# B&R Automation Studio project dbserv_0640
Automation Studio 6.5.3.11

## Configuration CP3686X

CPU X20CP3686X, AutomationRuntime 6.7.6, Build 11.3.0

### Task classes (Cpu.sw)
```
Cyclic#3:
  io <- IO-Treiber.io.prg
  kupplung <- Anwendung.kupplung.prg
  anlage <- Anwendung.anlage.prg
  iec103 <- IEC103-Treiber.iec103.prg
  iodrv <- IO-Treiber.iodrv.prg
  dbsevent <- DbServ-Basis.dbsevent.prg
  iec103Cmd <- IEC103-Treiber.iec103Cmd.prg
Cyclic#4:
  def <- def.prg
  Lebensbit <- Lebensbit.prg
  zaehler <- zaehler.prg
Cyclic#8:
  dbstcp <- DbServ-Basis.dbstcp.prg
  dbserv <- DbServ-Basis.dbserv.prg
  dbsmon <- DbServ-Basis.dbsmon.prg
  dbstest <- DbServ-Basis.dbstest.prg
DataObjects: dplist <- Anwendung.dplist.dob, typlist <- Anwendung.typlist.dob
Binaries: TCData, udbdef, sysconf, iomap, asfw, arconfig, ashwd, ashwac, mvLoader
Libraries: dbslib, sys_lib, standard, runtime, OPERATOR, FileIO, dvframe, DPMaster, DataObj, CAN_Lib, brsystem, astime, AsHW, AsBrStr, IEC103Ut, ArEventLog, AsIecCon, ethsock
```

### Hardware
```
PLC1 : X20CP3686X v1.10.0.0
  Connector IF2:
    ActivateDevice = 1
    HostName = audiinba6183
    Mode = Manual
    InternetAddress = 192.168.0.86
    SubnetMask = 255.255.255.0
    ActivateSnmp = 2
  Connector IF3:
    CycleTime = 2000
    InaPort = 11161
    InaNodeNumber = 0
  ConfigurationID = dbserv86_Config1
  UserPartitionSize = 0
  UserRamSize = 966656
  RemMemSize = 65280
  VolatileGlobalPvSize = 4096
  XLinkUseDefault = 0
  XLinkDuration = 10000
  FileDevice1
  FileDeviceName1 = USER
  FileDevicePath1 = USER_PATH
  EthernetHostName = DbServ
  EthernetDefaultGateway = 255.255.255.255
  ActivateWebServer = 0
  ActivateSdm = 0
  ActivateFtpServer = 1
X20BM11 : X20BM11 v1.1.0.0 (Disabled=true)  [X2X1 -> PLC1.IF6]
X20CS1030 : X20CS1030 v1.8.3.0 (Disabled=true)  [SS1 -> X20TB12.SS; SL -> X20BM11.SL1]
X20TB12 : X20TB12 v1.0.0.0 (Disabled=true)
```

### ACTIVE_GDM.osl - PLC1/States/ACTIVE_GDM.osl
```
ObjectStates:
  Object io (Memory=UserROM, Enable=true)
  Object zaehler (Memory=UserROM, Enable=false)
  Object kupplung (Memory=UserROM, Enable=true)
  Object iec103 (Memory=UserROM, Enable=true)
  Object iodrv (Memory=UserROM, Enable=true)
  Object l2dp (Memory=UserROM, Enable=true)
  Object dbsevent (Memory=UserROM, Enable=false)
  Object battery (Memory=UserROM, Enable=true)
  Object dbserv (Memory=UserROM, Enable=true)
  Object dbsmon (Memory=UserROM, Enable=true)
  Object dbstest (Memory=UserROM, Enable=false)
  Object dbstcp (Memory=UserROM, Enable=true)
  Object dbvist (Memory=UserROM, Enable=true)
  Object dbvisint (Memory=UserROM, Enable=true)
  Object gps (Memory=UserROM, Enable=true)
  Object version (Memory=UserROM, Enable=true)
  Object ydplist (Memory=UserROM, Enable=false)
  Object ytyplist (Memory=UserROM, Enable=false)
  Object dplist1 (Memory=UserROM, Enable=false)
  Object typlist1 (Memory=UserROM, Enable=false)
  Object dplist (Memory=UserROM, Enable=true)
  Object typlist (Memory=UserROM, Enable=true)
  Object dplisto (Memory=UserROM, Enable=false)
  Object ioimgcfg (Memory=UserROM, Enable=true)
  Object a_rflx_io (Memory=UserROM, Enable=true)
  Object dbv_text (Memory=UserROM, Enable=true)
  Object dbv_par (Memory=UserROM, Enable=true)
  Object dbv_env (Memory=UserROM, Enable=true)
  Object dbv_atoa (Memory=UserROM, Enable=true)
  Object dbv_func (Memory=UserROM, Enable=true)
  Object dbv_code (Memory=UserROM, Enable=true)
  Object dbv_rs (Memory=UserROM, Enable=true)
  Object dbv_vt1 (Memory=UserROM, Enable=true)
  Object dpm_099 (Memory=UserROM, Enable=true)
  Object sysconf (Memory=SystemROM, Enable=true)
  Object String_x (Memory=UserROM, Enable=true)
  Object megafubs (Memory=UserROM, Enable=true)
  Object dbv_lib (Memory=UserROM, Enable=true)
  Object dbvi_lib (Memory=UserROM, Enable=true)
  Object dbslib (Memory=UserROM, Enable=true)
  Object DA_x (Memory=UserROM, Enable=true)
```

## Logical view

Binary libraries used (declarations not repeated): ETHSOCK, sys_lib, runtime, standard, operator, FileIO, dvframe, DPMaster, DataObj, CAN_Lib, brsystem, astime, AsBrStr, AsHW, ArEventLog, AsIecCon

### Data object Logical/version (Simple, version 6.00.0) - Softwarestand

#### version.dat
```
; durchgeführte Software-Änderungen

;	14.07.2023	BIE     Version 6.40.0 		Kompiliert mit AS 4.12.3
;											für ATOM-CPUs mit AR E4.93

;	08.11.2021	BIE     Version 6.30.0 		Bugfix in Modul dbserv.c

;	15.07.2021	BIE     Version 6.20.0 		Kompiliert mit AS 4.9.3
;											für ATOM-CPUs mit AR D4.90
;											CELERON-CPUs werden nicht mehr unterstützt

;	02.03.2020	BIE     Version 6.11.0 		Kompiliert mit AS 4.6.4
;											für ATOM-CPUs mit AR C4.63
;											für CELERON-CPUs mit AR H3.10

;	04.12.2019	BIE     Version 6.10.0 		Kompiliert mit AS 4.4.6
;											für ATOM-CPUs mit AR C4.45
;											Lib IEC103Ut für IEC-Kommandos wurde hinzugefügt
;											dbseventtreiber aktualisiert
;
;	08.03.2019	BIE     Version 6.00.0 		Kompiliert mit AS 4.4.6
;											für ATOM-CPUs mit AR G4.34
;
;   12.10.2016	BIE     Version 4.11.0 		Kompiliert mit AS 4.1.11
;											Der angepasste IEC-Treiber von WAI wurde hinzugefügt und der dbsevent Treiber von KRZ
;											Ausserdem werden nun zwei Versionen der .br-Module veröffentlicht:
;											4.11.0 für ATOM-CPUs mit AR E4.10
;											3.11.0 für ATOM-CPUs mit AR V3.09

;   31.07.15	BIE     Version 4.10.0 		Portierung in AS 4.1.6.81 mit AR E4.10
;											inkl. Anpassungen für dbtcp für ATOM CPUs mit AR >x4.xx
;
;	12.08.13	WAI		Version 3.00.0		diverse Tests, Bereinigung der Sourcecodes
;
;	29.07.13	KRZ		Version 3.00.0		Portierung auf AS 3.0.90.23 SP05
;
;	30.06.11	RES		Version 2.07.1		Entwicklungsprojekt und Beispielprojekt mit AS2.7 kompiliert
;											AS V 2.7.0.20 SP13
;											AR N 2.95
;											Keine funktionellen Aenderungen
;
;	18.01.11	RES		Version 2.07		Erste freigegebene Vollversion für X20 CPUs
;						dbserv86.pgp		Neues Entwicklungsprojekt mit X20CP3486 erstellt
;											AS V 2.6.0.7
;											AR V 2.92
;						dbsbs486.pgp		Neues Beispielprojekt für X20CP3486 erstellt
;											AS + AR wie oben
;											Keine funktionellen Aenderungen
;
;	26.11.10	WAI		Version 2.06.4
;						iec103		IsANumber() geaendert: nun mit Vorzeichen Unterstuetzung
;						iodrv		Schreibzugriff auf PVs aktiviert
;
;	04.11.09	WAI		Version 2.06.3
;						l2dp		um510.c	verbesserte Reihenfolge beim Polling der Profile wegen Probleme bei langsamen Reaktionszeiten
;
;	12.10.09	WAI		Version 2.06.2
;						l2dp		neues Schlüsselwort Endian (=Big oder =Little) für Byte-Order
;									Profibus-Diagnose pL2DP_PbDataIn jetzt 244 statt 128 Byte
;
;	01.10.09	WAI		Version 2.06.1
;						l2dp		neues Schlüsselwort Inv (Invers) für BOOL-Variablen
;
;	21.08.09	WAI		Version 2.06 alle Module gestempelt
;						l2dp		neue Device-Variante UMG510
;									neue Schlüsselworte für GSD-Treiber (Mode, ModePar) wegen SYMAP
;
;	21.04.08	WAI		Version 2.05
;						l2dp		neue Device-Variante SPAZC302 für ABB-Gateways
;
;	20.02.08	WAI		Version 2.04
;						l2dp		neue Device-Variante UMGProfil für UMG96S und UMG507
;
;	28.01.08	RES		Version 2.04
;						dbslib:		Fehlerbehebung durch KUR: Status bei DbsGetBool() und DbsGetInt()
;						dbvi_lib:	Fehlerbehebung durch KUR: Output-Aktualisierung in letzter Displayzeile
;
;	25.06.07	WAI		Version 2.03 für IEC-Treiber (Anpassung Mode 13)
;
;	18.05.07	WAI		Version 2.02
;						dbsmon.c	Anzeige des valid-Status
;						gsd.c,l2dp.h,l2dp_parse.c,l2dp_parse.h
;									neuer Profibus-Typ "GSD"
;									jetzt 4 statt 1 L2DP-Linie möglich, dafür aber max. 64 statt 128 devices per line
;									(wegen 64kB-Grenze)
;						dbv_text.dat negative Werte ermöglicht incl. Korrektur bei Nachkommastellen
;						dbvist.c	Alarmquittierung aktiviert (direktes Schreiben in PAB)
;						alle anderen Module:	ebenfalls auf V2.02 gestempelt, um Verwirrungen zu vermeiden
;
;	09.05.07	WAI		Version 2.01 (Projektabgleich)
;						l2dp.c		Defaultwert Fakt = 1.0
;						umg503.c	kein neuer Request bei Kopplungsstörung wegen wiederholten Fehlermeldungen
;						iodrv.c		Schreibattribut für quittierpflichtige Variablen
;						dbv_rs.dat	9600Bd wegen Problem mit IF060 und Tableau
;
;	08.09.06	WAI		Version 2.00
;	04.07.06	WAI		Version mit neuem DbVist
;	22.06.06	WAI		Version mit DbVist
;	07.04.06	WAI		Erstfassung
```

### Global.typ
```iecst
TYPE
	XstDiagnose : 	STRUCT
		ulFRM_rbufFailAnz : UDINT;
		ulFRM_readFailAnz : UDINT;
		ulWrongTelAnz : UDINT;
		ulDTExSetTimeFail : UDINT;
		ulTelTimeoutAnz : UDINT;
		ulSyncAnz : UDINT;
		ulRTC_gettimeFail : UDINT;
		ulSyncPosFail : UDINT;
	END_STRUCT;
	XstMeinberg : 	STRUCT
		ucTag : USINT;
		ucMonat : USINT;
		ucJahr : USINT;
		ucStunden : USINT;
		ucMinuten : USINT;
		ucSekunden : USINT;
		ucSyncOK : USINT;
		ucPosOK : USINT;
		ucZZone : USINT;
		ucZSprung : USINT;
	END_STRUCT;
END_TYPE
```

### Library Logical/Libraries/IEC103Ut (IEC, version 6.40.0)

#### IEC103Ut.typ - Exported data types
```iecst
TYPE
	IEC103Ut_WrCmd_PVInfo_Type : 	STRUCT
		PVAdr : UDINT;
		PVLen : UDINT;
		PVDataType : UDINT;
		PVDimension : UINT;
	END_STRUCT;
END_TYPE
```

#### IEC103Ut.var - Exported constants
```iecst
VAR CONSTANT
	IEC103Ut_DATA_TYPE_STRUCT : USINT := 0;
	IEC103Ut_DATA_TYPE_STRUCT_2 : USINT := 15;
	IEC103Ut_DATA_TYPE_BOOL : USINT := 1;
	IEC103Ut_DATA_TYPE_SINT : USINT := 2;
	IEC103Ut_DATA_TYPE_INT : USINT := 3;
	IEC103Ut_DATA_TYPE_DINT : USINT := 4;
	IEC103Ut_DATA_TYPE_USINT : USINT := 5;
	IEC103Ut_DATA_TYPE_UINT : USINT := 6;
	IEC103Ut_DATA_TYPE_UDINT : USINT := 7;
	IEC103Ut_DATA_TYPE_REAL : USINT := 8;
	IEC103Ut_DATA_TYPE_STRING : USINT := 9;
	IEC103Ut_DATA_TYPE_ULINT : USINT := 10;
	IEC103Ut_DATA_TYPE_DATE_AND_TIME : USINT := 11;
	IEC103Ut_DATA_TYPE_TIME : USINT := 12;
	IEC103Ut_DATA_TYPE_DATE : USINT := 13;
	IEC103Ut_DATA_TYPE_LREAL : USINT := 14;
END_VAR
(**)
VAR CONSTANT
	IEC103Ut_FUB_IDLE : DINT := 65533;
	IEC103Ut_FUB_DISABLED : DINT := 65534;
	IEC103Ut_FUB_BUSY : DINT := 65535;
	IED103Ut_ERROR_START : DINT := 50000;
	IED103Ut_ERROR_INPUT_INVALID : DINT := IED103Ut_ERROR_START+2000;
END_VAR
```

#### IEC103Ut.fun - Exported functions and function blocks
```iecst
{REDUND_ERROR} FUNCTION_BLOCK IEC103Ut_WrCmd (*TODO: Hier einen Kommentar eingeben*) (*$GROUP=User,$CAT=User,$GROUPICON=User.png,$CATICON=User.png*)
	VAR_INPUT
		Enable : BOOL;
		DataSend : BOOL;
		LineVarStr : UDINT;
		LineNumber : USINT;
		DeviceAdr : USINT;
		FunctionType : USINT;
		InformationNumber : USINT;
		Val : USINT;
	END_VAR
	VAR_OUTPUT
		Status : DINT;
	END_VAR
	VAR
		WrCmdStep : UINT;
		PVStr : STRING[100];
		ValStr : STRING[10];
		ItemStr : STRING[100];
		PV_xgetadr_status : UINT;
		PV_ninfo_status : UINT;
		PVInfo_AnlStruct : IEC103Ut_WrCmd_PVInfo_Type;
		PVInfo_AnlStructOld : IEC103Ut_WrCmd_PVInfo_Type;
		PVInfo_DataSend : IEC103Ut_WrCmd_PVInfo_Type;
		PVInfo_DeviceAdress : IEC103Ut_WrCmd_PVInfo_Type;
		PVInfo_FunctionType : IEC103Ut_WrCmd_PVInfo_Type;
		PVInfo_InformationNumber : IEC103Ut_WrCmd_PVInfo_Type;
		PVInfo_Val : IEC103Ut_WrCmd_PVInfo_Type;
		PVInfo_Ready : IEC103Ut_WrCmd_PVInfo_Type;
		PVInfo_Error : IEC103Ut_WrCmd_PVInfo_Type;
		IECIEC103Ut_WrSimplePV_0 : IEC103Ut_WrSimplePV;
		IEC103Ut_RdSimplePV_0 : IEC103Ut_RdSimplePV;
		LineVarStrOld : UDINT;
		LineNumberOld : USINT;
	END_VAR
END_FUNCTION_BLOCK

{REDUND_ERROR} FUNCTION_BLOCK IEC103Ut_WrSimplePV (*TODO: Hier einen Kommentar eingeben*) (*$GROUP=User,$CAT=User,$GROUPICON=User.png,$CATICON=User.png*)
	VAR_INPUT
		PVAdr : {REDUND_UNREPLICABLE} UDINT;
		DataType : UDINT;
		PVValue : DINT;
	END_VAR
	VAR_OUTPUT
		valid : BOOL;
	END_VAR
	VAR
		pPV_BOOL : REFERENCE TO BOOL;
		pPV_USINT : REFERENCE TO USINT;
		pPV_UINT : REFERENCE TO UINT;
		pPV_UDINT : REFERENCE TO UDINT;
		pPV_SINT : REFERENCE TO SINT;
		pPV_INT : REFERENCE TO INT;
		pPV_DINT : REFERENCE TO DINT;
		pPV_REAL : REFERENCE TO REAL;
	END_VAR
END_FUNCTION_BLOCK

{REDUND_ERROR} FUNCTION_BLOCK IEC103Ut_RdSimplePV (*TODO: Hier einen Kommentar eingeben*) (*$GROUP=User,$CAT=User,$GROUPICON=User.png,$CATICON=User.png*)
	VAR_INPUT
		PVAdr : {REDUND_UNREPLICABLE} UDINT;
		DataType : UDINT;
	END_VAR
	VAR_OUTPUT
		PVValue : DINT;
		valid : BOOL;
	END_VAR
	VAR
		pPV_BOOL : REFERENCE TO BOOL;
		pPV_USINT : REFERENCE TO USINT;
		pPV_UINT : REFERENCE TO UINT;
		pPV_UDINT : REFERENCE TO UDINT;
		pPV_SINT : REFERENCE TO SINT;
		pPV_INT : REFERENCE TO INT;
		pPV_DINT : REFERENCE TO DINT;
		pPV_REAL : REFERENCE TO REAL;
	END_VAR
END_FUNCTION_BLOCK
```

#### IEC103Ut_WrCmd.st
```iecst
(*
-----------------------------------------------
FUNCTION Block IEC103Ut_WrCmd

	Write commands to a device, using the command structure OF IEC103 Task

	Inputs:
		Enable		 		Enable function block
		DataSend			Send command do device (edge sensitive)
		LineVarStr			Option: Adress OF name OF local PV structure element in Task IEC103 (example: "iec103:stANL[0].Command")
		LineNumber			Option:	Linenumber (1..12)
							Either LineVarStr or LineNumber is necessary
		DeviceAdr			Adress of device
		FunctionType		Function Type
		InformationNumber	Information Number
		Val					Value

	Outputs:
		Status				0 		Function ready, without error

							52000	Invalid input parameter
							52008	Timeout response telegram
							52020	command NOT accepted
							52023	response telegram: value not equal
							52024	response telegram: return information not equal
							52025	command function disabled
							52026	connection to device not ready
							52027	wrong device adress
							52028	command function still active

							3300 - 14714	error state of function PV_xgetadr or PV_ninfo (see B&R Help)

							65533	functionblock idle
							65534	functionblock disabled
							65535	functionblock busy

	Version:
	07.02.2019	Version 1.0
				first edition

-----------------------------------------------
*)
FUNCTION_BLOCK IEC103Ut_WrCmd

	IF(Enable = TRUE) THEN
		CASE WrCmdStep OF
			0:
				// ---------------------
				// check input parameter
				IF((LineVarStr = 0) AND (LineNumber = 0)) THEN
					Status		:= IED103Ut_ERROR_INPUT_INVALID;
					WrCmdStep	:= 210;
				ELSE

					Status := IEC103Ut_FUB_BUSY;
					// ---------------------------------------------
					// get name and adress of main structure element
					IF(LineVarStr = 0) THEN
						// Adresse der Anlagenstruktur ermitteln: PV Name erzeugen und PV Adresse ermitteln
						brsstrcpy(ADR(PVStr),ADR('iec103:stANL['));
						brsitoa(USINT_TO_DINT(LineNumber-1),ADR(ValStr));
						brsstrcat(ADR(PVStr),ADR(ValStr));
						brsstrcat(ADR(PVStr),ADR('].Command'));
					ELSE
						// Adresse der Anlagenstruktur ermitteln: Uebergebenen PV Namen verwenden und PV Adresse ermitteln
						brsstrcpy(ADR(PVStr),LineVarStr);
					END_IF

					PV_xgetadr_status := PV_xgetadr(ADR(PVStr),ADR(PVInfo_AnlStruct.PVAdr),ADR(PVInfo_AnlStruct.PVLen));

					IF(PV_xgetadr_status = 0) THEN
						LineNumberOld	:= LineNumber;
						LineVarStrOld	:= LineVarStr;
						WrCmdStep		:= 10;
					ELSE
						Status			:= PV_xgetadr_status;
						WrCmdStep		:= 210;
					END_IF
				END_IF

			10:	// get adress and info about structure element: DataSend
				brsstrcpy(ADR(ItemStr),ADR(PVStr));
				brsstrcat(ADR(ItemStr),ADR('.DataSend'));
				PV_xgetadr_status := PV_xgetadr(ADR(ItemStr),ADR(PVInfo_DataSend.PVAdr),ADR(PVInfo_DataSend.PVLen));
				IF(PV_xgetadr_status = 0) THEN
					WrCmdStep	:= 11;
				ELSE
					Status		:= PV_xgetadr_status;
					WrCmdStep	:= 210;
				END_IF

			11:
				PV_ninfo_status := PV_ninfo(ADR(ItemStr),ADR(PVInfo_DataSend.PVDataType),ADR(PVInfo_DataSend.PVLen),ADR(PVInfo_DataSend.PVDimension));
				IF(PV_ninfo_status = 0) THEN
					WrCmdStep	:= 15;
				ELSE
					Status		:= PV_ninfo_status;
					WrCmdStep	:= 210;
				END_IF

			15:	// get adress and info about structure element: PVInfo_DeviceAdress
				brsstrcpy(ADR(ItemStr),ADR(PVStr));
				brsstrcat(ADR(ItemStr),ADR('.DeviceAdress'));
				PV_xgetadr_status := PV_xgetadr(ADR(ItemStr),ADR(PVInfo_DeviceAdress.PVAdr),ADR(PVInfo_DeviceAdress.PVLen));
				IF(PV_xgetadr_status = 0) THEN
					WrCmdStep	:= 16;
				ELSE
					Status		:= PV_xgetadr_status;
					WrCmdStep	:= 210;
				END_IF

			16:
				PV_ninfo_status := PV_ninfo(ADR(ItemStr),ADR(PVInfo_DeviceAdress.PVDataType),ADR(PVInfo_DeviceAdress.PVLen),ADR(PVInfo_DeviceAdress.PVDimension));
				IF(PV_ninfo_status = 0) THEN
					WrCmdStep	:= 20;
				ELSE
					Status		:= PV_ninfo_status;
					WrCmdStep	:= 210;
				END_IF

			20:	// get adress and info about structure element: FunctionType
				brsstrcpy(ADR(ItemStr),ADR(PVStr));
				brsstrcat(ADR(ItemStr),ADR('.FunctionType'));
				PV_xgetadr_status := PV_xgetadr(ADR(ItemStr),ADR(PVInfo_FunctionType.PVAdr),ADR(PVInfo_FunctionType.PVLen));
				IF(PV_xgetadr_status = 0) THEN
					WrCmdStep	:= 21;
				ELSE
					Status		:= PV_xgetadr_status;
					WrCmdStep	:= 210;
				END_IF

			21:
				PV_ninfo_status := PV_ninfo(ADR(ItemStr),ADR(PVInfo_FunctionType.PVDataType),ADR(PVInfo_FunctionType.PVLen),ADR(PVInfo_FunctionType.PVDimension));
				IF(PV_ninfo_status = 0) THEN
					WrCmdStep	:= 25;
				ELSE
					Status		:= PV_ninfo_status;
					WrCmdStep	:= 210;
				END_IF

			25:	// get adress and info about structure element: InformationNumber
				brsstrcpy(ADR(ItemStr),ADR(PVStr));
				brsstrcat(ADR(ItemStr),ADR('.InformationNumber'));
				PV_xgetadr_status := PV_xgetadr(ADR(ItemStr),ADR(PVInfo_InformationNumber.PVAdr),ADR(PVInfo_InformationNumber.PVLen));
				IF(PV_xgetadr_status = 0) THEN
					WrCmdStep	:= 26;
				ELSE
					Status		:= PV_xgetadr_status;
					WrCmdStep	:= 210;
				END_IF

			26:
				PV_ninfo_status := PV_ninfo(ADR(ItemStr),ADR(PVInfo_InformationNumber.PVDataType),ADR(PVInfo_InformationNumber.PVLen),ADR(PVInfo_InformationNumber.PVDimension));
				IF(PV_ninfo_status = 0) THEN
					WrCmdStep	:= 30;
				ELSE
					Status		:= PV_ninfo_status;
					WrCmdStep	:= 210;
				END_IF

			30:	// get adress and info about structure element: Val
				brsstrcpy(ADR(ItemStr),ADR(PVStr));
				brsstrcat(ADR(ItemStr),ADR('.Val'));
				PV_xgetadr_status := PV_xgetadr(ADR(ItemStr),ADR(PVInfo_Val.PVAdr),ADR(PVInfo_Val.PVLen));
				IF(PV_xgetadr_status = 0) THEN
					WrCmdStep	:= 31;
				ELSE
					Status		:= PV_xgetadr_status;
					WrCmdStep	:= 210;
				END_IF

			31:
				PV_ninfo_status := PV_ninfo(ADR(ItemStr),ADR(PVInfo_Val.PVDataType),ADR(PVInfo_Val.PVLen),ADR(PVInfo_Val.PVDimension));
				IF(PV_ninfo_status = 0) THEN
					WrCmdStep	:= 35;
				ELSE
					Status		:= PV_ninfo_status;
					WrCmdStep	:= 210;
				END_IF

			35:	// get adress and info about structure element: Ready
				brsstrcpy(ADR(ItemStr),ADR(PVStr));
				brsstrcat(ADR(ItemStr),ADR('.Ready'));
				PV_xgetadr_status := PV_xgetadr(ADR(ItemStr),ADR(PVInfo_Ready.PVAdr),ADR(PVInfo_Ready.PVLen));
				IF(PV_xgetadr_status = 0) THEN
					WrCmdStep	:= 36;
				ELSE
					Status		:= PV_xgetadr_status;
					WrCmdStep	:= 210;
				END_IF

			36:
				PV_ninfo_status := PV_ninfo(ADR(ItemStr),ADR(PVInfo_Ready.PVDataType),ADR(PVInfo_Ready.PVLen),ADR(PVInfo_Ready.PVDimension));
				IF(PV_ninfo_status = 0) THEN
					WrCmdStep	:= 40;
				ELSE
					Status		:= PV_ninfo_status;
					WrCmdStep	:= 210;
				END_IF

			40:	// get adress and info about structure element: Error
				brsstrcpy(ADR(ItemStr),ADR(PVStr));
				brsstrcat(ADR(ItemStr),ADR('.Error'));
				PV_xgetadr_status := PV_xgetadr(ADR(ItemStr),ADR(PVInfo_Error.PVAdr),ADR(PVInfo_Error.PVLen));
				IF(PV_xgetadr_status = 0) THEN
					WrCmdStep	:= 41;
				ELSE
					Status		:= PV_xgetadr_status;
					WrCmdStep	:= 210;
				END_IF

			41:
				PV_ninfo_status := PV_ninfo(ADR(ItemStr),ADR(PVInfo_Error.PVDataType),ADR(PVInfo_Error.PVLen),ADR(PVInfo_Error.PVDimension));
				IF(PV_ninfo_status = 0) THEN
					WrCmdStep	:= 100;
				ELSE
					Status		:= PV_ninfo_status;
					WrCmdStep	:= 210;
				END_IF

			100:
				// Idle step, wait for command to send
				IF(DataSend = TRUE) THEN
					IF((LineNumberOld <> LineNumber) OR (LineVarStrOld <> LineVarStr)) THEN
						Status		:= IEC103Ut_FUB_BUSY;
						WrCmdStep	:= 0;
					ELSE
						IF(DeviceAdr = 0) THEN
							Status		:= IED103Ut_ERROR_INPUT_INVALID;
							WrCmdStep	:= 120;
						ELSE
							// Send command to device
							Status := IEC103Ut_FUB_BUSY;

							// Write parameter and command to local structure of iec task
							IECIEC103Ut_WrSimplePV_0(PVAdr := PVInfo_Ready.PVAdr, 				DataType := PVInfo_Ready.PVDataType,				PVValue := 0);
							IECIEC103Ut_WrSimplePV_0(PVAdr := PVInfo_FunctionType.PVAdr,		DataType := PVInfo_FunctionType.PVDataType,			PVValue := FunctionType);
							IECIEC103Ut_WrSimplePV_0(PVAdr := PVInfo_InformationNumber.PVAdr,	DataType := PVInfo_InformationNumber.PVDataType,	PVValue := InformationNumber);
							IECIEC103Ut_WrSimplePV_0(PVAdr := PVInfo_Val.PVAdr,					DataType := PVInfo_Val.PVDataType,					PVValue := Val);
							IECIEC103Ut_WrSimplePV_0(PVAdr := PVInfo_DeviceAdress.PVAdr,		DataType := PVInfo_DeviceAdress.PVDataType,			PVValue := DeviceAdr);
							IECIEC103Ut_WrSimplePV_0(PVAdr := PVInfo_DataSend.PVAdr,			DataType := PVInfo_DataSend.PVDataType,				PVValue := 1);
							WrCmdStep		:= 110;
						END_IF
					END_IF
				ELSE
					Status	:= IEC103Ut_FUB_IDLE;
				END_IF

			110:
				// Read result information from local structure of iec task
				IEC103Ut_RdSimplePV_0(PVAdr := PVInfo_Ready.PVAdr, DataType := PVInfo_Ready.PVDataType);

				// Ready
				IF(IEC103Ut_RdSimplePV_0.PVValue > 0) THEN
					// Error Information
					IEC103Ut_RdSimplePV_0(PVAdr := PVInfo_Error.PVAdr, DataType := PVInfo_Error.PVDataType);
					IF(IEC103Ut_RdSimplePV_0.PVValue = 0) THEN
						Status	:= 0;
					ELSE
						Status	:= IED103Ut_ERROR_START + DINT_TO_UINT(IEC103Ut_RdSimplePV_0.PVValue);
					END_IF
					WrCmdStep	:= 120;
				END_IF

				IF(DataSend = FALSE) THEN
					Status		:= IEC103Ut_FUB_IDLE;
					WrCmdStep	:= 100;
				END_IF

			120:
				// Wait until command is cleared
				IF(DataSend = FALSE) THEN
					Status		:= IEC103Ut_FUB_IDLE;
					WrCmdStep	:= 100;
				END_IF

			210:
				// Error Step, function block has to be disabled
		END_CASE
	ELSE
		WrCmdStep	:= 0;
		Status		:= IEC103Ut_FUB_DISABLED;
	END_IF

END_FUNCTION_BLOCK
```

#### IEC103Ut_WrSimplePV.st
```iecst
(*
-----------------------------------------------
FUNCTION Block IEC103Ut_WrSimplePV

	Write value of a PV

	Inputs:
		PVAdr				Adress of PV
		DataType			Datatype of PV
		PVValue				Value witch is written

	Outputs:
		valid				TRUE	Datatype valid
							FALSE	Adress of PV or Datatype not valid

	Version:
	07.02.2019	Version 1.0
				first edition

-----------------------------------------------
*)
FUNCTION_BLOCK IEC103Ut_WrSimplePV

	valid := TRUE;

	IF(PVAdr <> 0) THEN
		CASE DataType OF

			IEC103Ut_DATA_TYPE_BOOL:
				pPV_BOOL ACCESS PVAdr;
				pPV_BOOL := DINT_TO_BOOL(PVValue);

			IEC103Ut_DATA_TYPE_USINT:
				pPV_USINT ACCESS PVAdr;
				pPV_USINT := DINT_TO_USINT(PVValue);

			IEC103Ut_DATA_TYPE_UINT:
				pPV_UINT ACCESS PVAdr;
				pPV_UINT := DINT_TO_UINT(PVValue);

			IEC103Ut_DATA_TYPE_UDINT:
				pPV_UDINT ACCESS PVAdr;
				pPV_UDINT := DINT_TO_UDINT(PVValue);

			IEC103Ut_DATA_TYPE_SINT:
				pPV_SINT ACCESS PVAdr;
				pPV_SINT := DINT_TO_SINT(PVValue);

			IEC103Ut_DATA_TYPE_INT:
				pPV_INT ACCESS PVAdr;
				pPV_INT := DINT_TO_INT(PVValue);

			IEC103Ut_DATA_TYPE_DINT:
				pPV_DINT ACCESS PVAdr;
				pPV_DINT := PVValue;
			ELSE
				valid:= FALSE;
		END_CASE
	ELSE
		valid:= FALSE;
	END_IF

END_FUNCTION_BLOCK
```

#### IEC103Ut_RdSimplePV.st
```iecst
(*-----------------------------------------------
FUNCTION Block IEC103Ut_RdSimplePV

	Read value of a PV

	Inputs:
		PVAdr				Adress OF PV
		DataType			Datatype OF PV

	Outputs:
		PVValue				Value of the PV
		valid				TRUE	Datatype valid
							FALSE	Adress OF PV OR Datatype NOT valid

	Version:
		07.02.2019	Version 1.0
		first edition

-----------------------------------------------
*)

FUNCTION_BLOCK IEC103Ut_RdSimplePV
	valid := TRUE;

	IF(PVAdr <> 0) THEN
		CASE DataType OF

			IEC103Ut_DATA_TYPE_BOOL:
				pPV_BOOL ACCESS PVAdr;
				PVValue := BOOL_TO_DINT(pPV_BOOL);

			IEC103Ut_DATA_TYPE_USINT:
				pPV_USINT ACCESS PVAdr;
				PVValue := USINT_TO_DINT(pPV_USINT);

			IEC103Ut_DATA_TYPE_UINT:
				pPV_UINT ACCESS PVAdr;
				PVValue := UINT_TO_DINT(pPV_UINT);

			IEC103Ut_DATA_TYPE_UDINT:
				pPV_UDINT ACCESS PVAdr;
				PVValue := UDINT_TO_DINT(pPV_UDINT);

			IEC103Ut_DATA_TYPE_SINT:
				pPV_SINT ACCESS PVAdr;
				PVValue := SINT_TO_DINT(pPV_SINT);

			IEC103Ut_DATA_TYPE_INT:
				pPV_INT ACCESS PVAdr;
				PVValue := INT_TO_DINT(pPV_INT);

			IEC103Ut_DATA_TYPE_DINT:
				pPV_DINT ACCESS PVAdr;
				PVValue := pPV_DINT;

			ELSE
				valid:= FALSE;
		END_CASE
	ELSE
		valid:= FALSE;
	END_IF
END_FUNCTION_BLOCK
```

### bksys.h
```c
/* bksys.h
// Globale Include-Datei fuer BURKLIMAT2000
// LastEdit:
//		14.08.03/RES:	bksys.h aus bk.h und bkklib.h erzeugt; neu in V4.01
//		12.08.03/RES:	Pipe-Diagnosen fuer Clients eingebaut; neu in V4.01
//		08.08.03/RES:	CliPipeItemLen aus DtProps_Typ entfernt ( wird nicht mehr benötigt )
//		06.08.03/RES:	ANZ_WAIT_CYCLE_xxx ueberarbeitet
//		18.07.03/RES:	Erweiterungen fuer V4.01 eingefuegt
//		05.06.03/RES:	Funktionsprototypen fuer Client-Interface eingefuegt
//		25.04.03/RES:	Erweiterungen fuer V4.00 eingefuegt
//		24.04.03/RES:	Basis-Fehlernummer von 60000 auf 50000 (=Anwenderbereich) geaendert
//		29.04.03/RES:	DtDesc.ItemOffPab von USINT auf USHORT geaendert ( wegen pCAB gab's Ueberlauf bei BKZS )
//		23.04.03/RES:	Datentypen für Client-Abbild (CAB) erweitert
//		22.04.03/RES:	Itemanzahlen (Bk2000) korrigiert!!
// --------------------------------------------- */

#ifndef BKSYS_H_
#define BKSYS_H_

/* Burklimat2000 - Versionsnummer fuer alle Bk2-Tasks */
#define BK_VERSION_NR			600			/* Vollversion=positiv, Betaversion=negativ */
#define BK_VERSION_TEXT			"V6.00.0"	/* Vollversion="V....", Betaversion="B...." */

/* Basis-Fehlernummer für Logbuch-Einträge */
#define EC_BK2_BASE				50000

/* Definitionen fuer Systemfunktionen */
#define EC_SYS_BASE				0
#define ERR_SYS_PRE				"bks"

/* Definitionen fuer bkfbklib */
#define EC_FBK_BASE				20
/* hier kein gemeinsames Prefix; jeder FBK hat eigenes Prefix!! */

/* Definitionen fuer bkkern */
#define EC_KERN_BASE			50
#define ERR_KERN_PRE			"bkk"

/* Definitionen fuer bkvist */
#define EC_VIST1_BASE			100			/* Pei 12.04.02 */
#define ERR_VIST1_PRE			"bkv"
#define ANZ_WAIT_CYCLE_VIST1	ANZ_WAIT_CYCLE_INET + 1

/* Definitionen fuer bkvist2 */
#define EC_VIST2_BASE			150
#define ERR_VIST2_PRE			"bkw"		/* von "bkv2" -> "bkw" geaendert: 22.05.02/RES */
#define ANZ_WAIT_CYCLE_VIST2	ANZ_WAIT_CYCLE_VIST1 + 5

/* Definitionen fuer bkinet */
#define EC_INET_BASE			200
#define ERR_INET_PRE			"bki"
#define USER_ID_INET			1
#define ANZ_WAIT_CYCLE_INET		ANZ_WAIT_CYCLE_TCP + 2

/* Definitionen fuer bktcp */
#define EC_TCP_BASE				250
#define ERR_TCP_PRE				"bkt"
#define ANZ_WAIT_CYCLE_TCP		0

/* Definitionen fuer dbs */
#define EC_DBS_BASE				300
#define ERR_DBS_PRE				"dbs"
#define ANZ_WAIT_CYCLE_DBS		0

/* Anzahl Fehlerzaehler fuer ErrStatistics */
#define ERRCNTANZ				300

/* maximale Anzahl Fehlereintraege ins Logbuch beim Parsen */
#define PARS_ERR_MAXENTRIES		5

enum Elementarten { EA_RK, EA_SG, EA_AP, EA_SW, EA_ZL, EA_SB, EA_BP, EA_AL, EA_BA=10, EA_ANZ };
enum Datentypen { RK, SGST, SGQS, SGIN, AP, SW, ZL, SB, SBIM, SBKL, BP, AL, BA, STAT, ZS, DT_ANZ };

enum EvTyp { IMP, EXP };						/* Event-Typ: Implizit / Explizit */
enum ErrStat { WARN, ERR, ERRLOG, ERRLOGHALT };	/* Fehlerstati */

#define USR_ANZ_MAX		8		/* maximale Anzahl der DCS2000-User */
#define CLI_ANZ_MAX		8		/* maximale Anzahl der ZLT-Clients; neu in V4.00 */

#define DTNAMELEN		4
#define DPNAMELEN		32
#define ITEMNAMELEN		5

/* Fehlertexte und -nummern */
#define	NOVALIDSTATSPTR_TEXT	"SYS_Statistic n. gefunden"
#define	NOVALIDSTATSPTR_NUM		0

#define	PCREATEERR_TEXT			"Fehler beim Erzeugen der Event-Pipes"
#define	PCREATEERR_NUM			1

#define	ECREATEERR_TEXT			"Fehler beim Erzeugen der Event-Parameterblöcke"
#define	ECREATEERR_NUM			2

#define	NOVALIDGLOBPTR_TEXT		"Ungültige Adresse in SYS_pGlobals"
#define	NOVALIDGLOBPTR_NUM		3

#define	DTERR_TEXT				"DT-Index ungültig"
#define	DTERR_NUM				4

#define	DPERR_TEXT				"DP-Index ungültig"
#define	DPERR_NUM				5

#define	EVTYPERR_TEXT			"Eventtyp ungültig"
#define	EVTYPERR_NUM			6

#define	NOEVBLKERR_TEXT			"Kein Eventblock gefunden"
#define	NOEVBLKERR_NUM			7

/* Dimensionierung der Fehlermeldungen im Logbuch */
#define ERRTEXT_MAXLEN		31
#define ERRTEXT_MAXLINES	3
#define SEARCH_COUNT_MAX	6
#define CUT_SIGN			'~'

/* Itemanzahl jedes Datentyps ( BK2000 )*/
#define RK_DT_ITEMANZ	37
#define SGST_DT_ITEMANZ	23
#define SGQS_DT_ITEMANZ	25
#define SGIN_DT_ITEMANZ	25
#define AP_DT_ITEMANZ	13
#define SW_DT_ITEMANZ	13
#define ZL_DT_ITEMANZ	16
#define SB_DT_ITEMANZ	27
#define SBIM_DT_ITEMANZ	25
#define SBKL_DT_ITEMANZ	19
#define BP_DT_ITEMANZ	8
#define AL_DT_ITEMANZ	23
#define BA_DT_ITEMANZ	17
#define STAT_DT_ITEMANZ	14
#define ZS_DT_ITEMANZ	222

#define MAX_DT_ITEMANZ	ZS_DT_ITEMANZ	/* Maximale Itemanzahl für PabDefault */

/* Itemanzahl jeder Elementart (BK alt) */
#define	RK_EA_ITEMANZ	18
#define	SGST_EA_ITEMANZ	12
#define	SGQS_EA_ITEMANZ	12
#define	SGIN_EA_ITEMANZ	12
#define AP_EA_ITEMANZ	4
#define SW_EA_ITEMANZ	4
#define ZL_EA_ITEMANZ	5
#define SB_EA_ITEMANZ	4
#define SBIM_EA_ITEMANZ	4
#define SBKL_EA_ITEMANZ	4
#define BP_EA_ITEMANZ	1
#define AL_EA_ITEMANZ	4
#define BA_EA_ITEMANZ	1
#define STAT_EA_ITEMANZ	2
#define ZS_EA_ITEMANZ	1	/* Hier nur Dummy !! */

/* Byteanzahl jeder Elementart (BK alt ) */
#define	RK_EA_DATALEN	32
#define	SGST_EA_DATALEN	18
#define	SGQS_EA_DATALEN	18
#define	SGIN_EA_DATALEN	18
#define	AP_EA_DATALEN	7
#define	SW_EA_DATALEN	6
#define	ZL_EA_DATALEN	11
#define	SB_EA_DATALEN	4
#define	SBIM_EA_DATALEN	4
#define	SBKL_EA_DATALEN	4
#define	BP_EA_DATALEN	1
#define	AL_EA_DATALEN	4
#define	BA_EA_DATALEN	1
#define	STAT_EA_DATALEN	2
#define ZS_EA_DATALEN	1	/* Hier nur Dummy !! */

/* Anzahl DP-Events, die gleichzeitig in Eventpipe passen sollen */
#define RK_EP_ENTRIES	40
#define SGST_EP_ENTRIES	40
#define SGQS_EP_ENTRIES	40
#define SGIN_EP_ENTRIES	40
#define AP_EP_ENTRIES	100
#define SW_EP_ENTRIES	80
#define ZL_EP_ENTRIES	60
#define SB_EP_ENTRIES	40
#define SBIM_EP_ENTRIES	20
#define SBKL_EP_ENTRIES	20
#define BP_EP_ENTRIES	40
#define AL_EP_ENTRIES	80
#define BA_EP_ENTRIES	20
#define STAT_EP_ENTRIES	1	/* Hier nur Dummy !! */
#define ZS_EP_ENTRIES	1	/* Hier nur Dummy !! */

/* Berechnung der erforderlichen Puffergroesse fuer Pipes */
#define RK_EP_BUFSIZE	( RK_EP_ENTRIES   * ( sizeof( ItemAdr_Typ ) + RK_EA_DATALEN   + ( RK_EA_DATALEN   & 1 ) ) + 2 )
#define SGST_EP_BUFSIZE	( SGST_EP_ENTRIES * ( sizeof( ItemAdr_Typ ) + SGST_EA_DATALEN + ( SGST_EA_DATALEN & 1 ) ) + 2 )
#define SGQS_EP_BUFSIZE	( SGQS_EP_ENTRIES * ( sizeof( ItemAdr_Typ ) + SGQS_EA_DATALEN + ( SGQS_EA_DATALEN & 1 ) ) + 2 )
#define SGIN_EP_BUFSIZE	( SGIN_EP_ENTRIES * ( sizeof( ItemAdr_Typ ) + SGIN_EA_DATALEN + ( SGIN_EA_DATALEN & 1 ) ) + 2 )
#define AP_EP_BUFSIZE	( AP_EP_ENTRIES   * ( sizeof( ItemAdr_Typ ) + AP_EA_DATALEN   + ( AP_EA_DATALEN   & 1 ) ) + 2 )
#define SW_EP_BUFSIZE	( SW_EP_ENTRIES   * ( sizeof( ItemAdr_Typ ) + SW_EA_DATALEN   + ( SW_EA_DATALEN   & 1 ) ) + 2 )
#define ZL_EP_BUFSIZE	( ZL_EP_ENTRIES   * ( sizeof( ItemAdr_Typ ) + ZL_EA_DATALEN   + ( ZL_EA_DATALEN   & 1 ) ) + 2 )
#define SB_EP_BUFSIZE	( SB_EP_ENTRIES   * ( sizeof( ItemAdr_Typ ) + SB_EA_DATALEN   + ( SB_EA_DATALEN   & 1 ) ) + 2 )
#define SBIM_EP_BUFSIZE	( SBIM_EP_ENTRIES * ( sizeof( ItemAdr_Typ ) + SBIM_EA_DATALEN + ( SBIM_EA_DATALEN & 1 ) ) + 2 )
#define SBKL_EP_BUFSIZE	( SBKL_EP_ENTRIES * ( sizeof( ItemAdr_Typ ) + SBKL_EA_DATALEN + ( SBKL_EA_DATALEN & 1 ) ) + 2 )
#define BP_EP_BUFSIZE	( BP_EP_ENTRIES   * ( sizeof( ItemAdr_Typ ) + BP_EA_DATALEN   + ( BP_EA_DATALEN   & 1 ) ) + 2 )
#define AL_EP_BUFSIZE	( AL_EP_ENTRIES   * ( sizeof( ItemAdr_Typ ) + AL_EA_DATALEN   + ( AL_EA_DATALEN   & 1 ) ) + 2 )
#define BA_EP_BUFSIZE	( BA_EP_ENTRIES   * ( sizeof( ItemAdr_Typ ) + BA_EA_DATALEN   + ( BA_EA_DATALEN   & 1 ) ) + 2 )
#define STAT_EP_BUFSIZE	( STAT_EP_ENTRIES * ( sizeof( ItemAdr_Typ ) + STAT_EA_DATALEN + ( STAT_EA_DATALEN & 1 ) ) + 2 )
#define ZS_EP_BUFSIZE	( ZS_EP_ENTRIES   * ( sizeof( ItemAdr_Typ ) + ZS_EA_DATALEN   + ( ZS_EA_DATALEN   & 1 ) ) + 2 )

/* Berechnung der erforderlichen Blockgroesse fuer einen Event-Pipeblock */
#define EP_BUFSIZE ( RK_EP_BUFSIZE + SGST_EP_BUFSIZE + SGQS_EP_BUFSIZE + SGIN_EP_BUFSIZE + AP_EP_BUFSIZE + SW_EP_BUFSIZE + ZL_EP_BUFSIZE + SB_EP_BUFSIZE + SBIM_EP_BUFSIZE + SBKL_EP_BUFSIZE + BP_EP_BUFSIZE + AL_EP_BUFSIZE + BA_EP_BUFSIZE + STAT_EP_BUFSIZE + ZS_EP_BUFSIZE )
#define EP_BLOCKSIZE ( sizeof(EvPbHead_Typ) + ( DT_ANZ * sizeof(PipeHead_Typ) ) + EP_BUFSIZE )

/* Union fuer verschiedene Datentypen */
typedef union {
	long Long;
	unsigned long Ulong;
	short Short;
	unsigned short Ushort;
	char Char[4];
	unsigned char Uchar[4];
} VarData_Typ;

/* Item-Adresse */
typedef struct {
	unsigned short DpIdx;
	unsigned char ItemOff;
	unsigned char ItemLen;
} ItemAdr_Typ;

/* Item-Adresse fuer CAB */
typedef struct {
	unsigned short DpIdx;
	unsigned char ItemIdx;
	unsigned char ItemLen;
} CabItemAdr_Typ;

/* Pipe-Header */
typedef struct {
	unsigned char *pStart;
	unsigned char *pEnd;
	unsigned char *pWrite;
	unsigned char *pRead;
	unsigned char WriteFlag;
	unsigned char ReadFlag;
} PipeHead_Typ;

/* Pipeblock-Header fuer bkinet */
typedef struct EvPbHead {
	unsigned char	UserID;
	PipeHead_Typ	*pDtPipe[DT_ANZ];
	struct EvPbHead	*pNext;
} EvPbHead_Typ;

/* Pipe-Eintrag für ZLT-Clients (fuer alle Items gleich !) ; neu in V4.01 */
typedef struct CliPipeEntry {
	CabItemAdr_Typ	ItemAdr;
	unsigned long	ItemVal;
} CliPipeEntry_Typ;

/* Pipe-Header für ZLT-Clients ; neu in V4.01 */
typedef struct {
	CliPipeEntry_Typ	*pFirst;
	CliPipeEntry_Typ	*pLast;
	CliPipeEntry_Typ	*pWrite;
	CliPipeEntry_Typ	*pRead;
	unsigned char 		WriteFlag;
	unsigned char 		ReadFlag;
} CliPipeHead_Typ;

/* Pipeblock-Header für ZLT-Clients ; neu in V4.00 */
typedef struct CliPbHead {
	CliPipeHead_Typ		*pDtPipe[DT_ANZ];
} CliPbHead_Typ;

/* Alloc-Struktur fuer EvParaBlock-Speicherverwaltung */
typedef struct {
	unsigned char *pEvParBase;
	unsigned long lEvParLen;
	unsigned char *pEvParAct;
	unsigned long lEvParFree;
} EvAlloc_Typ;

/* Pab-Header */
typedef struct {
	unsigned char	*pDtBase[DT_ANZ];
	unsigned short 	DpAnz[DT_ANZ];
} PabHeader_Typ ;

/* Cab-Header ; neu in V4.00 */
typedef struct {
	unsigned short 	ClientAnz;					/* Anzahl Clients */
	unsigned char 	CliLogon[CLI_ANZ_MAX]; 		/* Logon-Flag fuer jeden Client */
	unsigned char	*pDtBase[DT_ANZ];			/* Zeiger auf Daten in CAB (je DT) */
	unsigned short 	DpAnz[DT_ANZ];				/* Anzahl DP-Eintraege in CAB (je DT) */
	CliPbHead_Typ	*pClientPb[CLI_ANZ_MAX];	/* Array mit Zeigern auf Client-Pipebloecke in CAB */
} CabHeader_Typ ;

/* CAB-Itemeintrag ; neu in V4.00 */
typedef struct {
	unsigned char 	Link; 		/* Link-Flag fuer dieses Item */
	unsigned char 	Force; 		/* Kennung fuer ueberfaelligen Event */
	unsigned long 	LastVal;	/* Zuletzt an Client gemeldeter Wert */
	unsigned long	Hyst;		/* Hysteresewert fuer Eventueberwachung */
} CabItemEntry_Typ ;

/* Datentyp-Eigenschaften */
typedef struct {
	unsigned char  DtName[DTNAMELEN + 1];
	unsigned char  DtMaxItemIdx;
	unsigned char  DtDataLen;
	unsigned char  Ea;
	unsigned char  EaMaxItemIdx;
	unsigned char  EaDataLen;
	unsigned char  ItemConvMaxIdx;
	unsigned short DtPabLen;
	unsigned char  DpNameOff;
	unsigned char  DtIdxOff;
	unsigned char  DpIdxOff;
	unsigned char  AliasPtrOff;
	unsigned char  PabPtrOffAlias;
	unsigned char  InitOffAlias;
	unsigned char  AlMkOffAlias;
	unsigned char  QuStOffAlias;
	unsigned char  Quit2OffAlias;
	unsigned char  HandOffAlias;
	unsigned char  HaufOffAlias;
	unsigned char  HzuOffAlias;
	unsigned char  IntOffAlias;
	unsigned char  IntUserLevel;
	unsigned short EvCtrlOff;
	unsigned char  EvUserOff;
	unsigned char  EvNextOff;
	unsigned char  EvParLen;
	unsigned short EpBufsize;
	unsigned char  CabItemAnz;		/* Anzahl Itemeintraege in CAB ; neu in V4.00 */
	unsigned char  CabItemEntryLen;	/* Laenge eines Itemeintrages in CAB ; neu in V4.00 */
	unsigned char  CabPtrOff;		/* Offset des CAB-Zeigers im PAB ; neu in V4.00 */
} DtProps_Typ;

/* Elementart-Deskriptor mit Infos zu jedem Ea-Item */
typedef struct {
	unsigned char	Offset;
	unsigned char	Byteanz;
} EaDesc_Typ;

/* Datentyp-Deskriptor mit Infos zu jedem Dt-Item */
typedef struct {
	unsigned char	ItemName[ITEMNAMELEN + 1];
	unsigned char	ItemOff;
	char 			ItemLen;
	unsigned char	EvParOff;
	unsigned short	ItemOffPab;		/* Item-Offset im PAB ( 0 = kein PAB-Item */
	short			ItemDefault;
	unsigned char 	ItemNrCab;	/* Item-Nummer in CAB ( 0 = kein CAB-Item ) ; neu in V4.00 */
} DtDesc_Typ;

/* Item-Konvertierungstabelle ( Offset -> ItemIndex ) */
typedef struct {
	char ItemBk;
	char ItemBk2;
} ItemConv_Typ;

/* Pipe-Diagnose fuer einen Client; neu in V4.01 */
typedef struct {
	unsigned long 		AnyPipeEntry;			/* Summenzaehler fuer alle erfolgreichen ClientPipe-Eintraege */
	unsigned long 		AnyPipeEntryPerSec;		/* Anzahl erfolgreicher ClientPipe-Eintraege pro Sekunde */
	unsigned long 		AnyPipeFull; 			/* Summenzaehler fuer alle ClientPipe-Vollmeldungen */
	unsigned long 		DtPipeFull[DT_ANZ]; 	/* Zaehler fuer ClientPipe-Vollmeldungen je Datentyp */
	unsigned char 		DtPipeUse[DT_ANZ];	 	/* Fuellstandsanzeige der Pipe in Prozent */
} CliPipeDiagOne_Typ;

/* Gemeinsame Pipe-Diagnose fuer alle Clients; neu in V4.01 */
typedef struct {
	unsigned short		Init;					/* Initialisierungs-Flag */
	unsigned long		EntryCount;				/* Summenzaehler fuer alle erfolgreichen ClientPipe-Eintraege aller Clients */
	unsigned long		EntryCountPerSec;		/* Anzahl erfolgreicher ClientPipe-Eintraege aller Clients pro Sekunde */
	unsigned short		FullClient;				/* Client, dem die zuletzt als voll erkannte Pipe gehoert */
	unsigned short		FullDt;					/* Datentyp, dessen Pipe zuletzt als voll erkannt wurde */
	unsigned long		FullCount;				/* Summenzaehler fuer alle ClientPipe-Vollmeldungen aller CLients */
	CliPipeDiagOne_Typ	Client[CLI_ANZ_MAX];
} CliPipeDiagAll_Typ;

/* Struktur fuer globale Informationen */
typedef struct {
	unsigned char			PabValid;					/* Kennung PAB gültig */
	PabHeader_Typ			*pPab;						/* Zeiger auf PAB */
	unsigned long			PabLen;						/* Länge PAB */
	CabHeader_Typ			*pCab;						/* Zeiger auf CAB ; neu in V4.00 */
	unsigned long			CabLen;						/* Länge des gesamten CAB ; neu in V4.00 */
	EvPbHead_Typ			*pEvPipes;					/* Zeiger auf Event-Pipes */
	EvAlloc_Typ				*pEvAlloc;					/* Zeiger auf Arrays mit Event-Alloc-Infos */
	DtProps_Typ				*pDtProps;					/* Zeiger auf Array mit Datentyp-Eigenschaften */
	EaDesc_Typ				*pEaDesc[DT_ANZ];			/* Array mit Zeigern auf Elementart-Deskriptoren */
	DtDesc_Typ				*pDtDesc[DT_ANZ];			/* Array mit Zeigern auf Datentyp-Deskriptoren */
	ItemConv_Typ			*pItemConv[DT_ANZ];			/* Array mit Zeigern auf Item-Konvertierungstabellen */
	char					*pCabItemConv[DT_ANZ];		/* Array mit Zeigern auf CAB-Item-Konvertierungstabellen */
	unsigned short			Count10ms;					/* 10ms-Takt-Zaehler */
	unsigned short			Count100ms;					/* 100ms-Takt-Zaehler */
	unsigned char			UstNr;						/* Unterstations-Nummer */
	unsigned char			Oertl;						/* Oertlich */
	unsigned char			SammH;						/* Sammelhand */
	unsigned char			KplSt;						/* Kopplungsstoerung */
	unsigned char			ALnLe;						/* Alarmliste nicht leer */
	unsigned char			AlUnq;						/* Mindestens 1 unquittierter Alarm */
	unsigned char			OertlBkvist;				/* Oertlich von bkvist */
	unsigned char			OertlFremd;					/* Oertlich von Fremd-Visu */
	CliPipeDiagAll_Typ		*pCliPipeDiag;				/* Zeiger auf Pipe-Diagnose fuer alle Clients */
} Globals_Typ;

typedef struct {
	unsigned char Jahr;
	unsigned char Mon;
	unsigned char Tag;
	unsigned char Std;
	unsigned char Min;
	unsigned char Sek;
	unsigned short Milli;
} Timestamp_Typ;

/* Struktur fuer Fehler-Statistik */
typedef struct {
	unsigned short	LastWarn;
	unsigned short	LastErr;
	unsigned short	Init;
	Timestamp_Typ	LastInit;
	unsigned short	ErrCount[ERRCNTANZ];
} Stats_Typ;

/* Input-Struktur fuer InitTabItem() */
typedef struct {
	unsigned char EaItemAnz;
	EaDesc_Typ *pEaDesc;
	unsigned char DtItemAnz;
	DtDesc_Typ *pDtDesc;
	void *pAlias;
	void *pPab;
	void *pEvPb;
	ItemConv_Typ *pItemConv;
	char *pCabItemConv;
} InitTabInfo_Typ;

/* prototypes */
/* fuer bksysall --------------- */
void ErrStatistics( unsigned char *pTaskName, unsigned char ErrStat, unsigned short ErrNum, unsigned long ErrInfo, unsigned char *pErrPre, unsigned char *pErrText );
void GetGlobalsPtr( Globals_Typ **ppGlobals );
unsigned long bin_to_bcd_8 (unsigned long value);

/* fuer bksystools ------------- */
short GetDpInfoDt( char *pDpName, unsigned char DtIdx, unsigned short *pDpIdx, unsigned char **ppAlias );

/* fuer bksysfbk --------------- */
void ErrStatisticsX( unsigned char *pTaskName, unsigned short *pErrMk, unsigned short ErrBit, unsigned short *pSyErr, unsigned char ErrStat1, unsigned char ErrStatN, unsigned short ErrNum, unsigned long ErrInfo, unsigned char *pErrPre, unsigned char *pErrText );
short GetPabValidPtr( unsigned char **ppPabValid );
short GetSysClockPtr( unsigned short **ppC10, unsigned short **ppC100 );
void UserEvents( unsigned char DtIdx, ItemAdr_Typ ItemAdr, unsigned char EvUserId,
				 unsigned char *pPab, unsigned char *pFlags, unsigned char *pEvPara,
				 unsigned char *pOldBuf, unsigned char *pNewBuf, unsigned short DpMsgLen,
				 unsigned short sItemIdxMax, DtDesc_Typ *pDtDesc, EaDesc_Typ *pEaDesc,
				 unsigned char dT, unsigned char *pErrPre, unsigned short *pErrMask, unsigned short *pSysErr );
short CheckItemEvent( char *pVal, char *pValOld, void *pEvPara, unsigned short sEvItemOff, short sDataFormat, unsigned char dT100ms );
short MinMaxLong( long *pVal, long lMin, long lMax );
short MinMaxShort( short *pVal, short sMin, short sMax );
void SetAllEvParaData( unsigned short sItemIdxMax, unsigned char *pPab, unsigned char *pEvPara, DtDesc_Typ *pDtDesc );
void SetEvParaData( unsigned short sItem, unsigned char *pPab, unsigned char *pEvPara, DtDesc_Typ *pDtDesc );
short CopyPabToElBuf( unsigned char *pBuf, ItemAdr_Typ *pAdr, unsigned char *pPab, unsigned short sItemIdxMax, EaDesc_Typ *pEaDesc, DtDesc_Typ *pDtDesc );
short Kennlinie( short X, short Xmin, short Xmax, short Ymin, short Ymax );
void CliEvents( unsigned char DtIdx, unsigned short DpIdx, unsigned char *pPab, CabItemEntry_Typ *pCab, DtProps_Typ *pDtProps, DtDesc_Typ *pDtDesc );
short PipeWrite( PipeHead_Typ* pPipe, unsigned char* pMsg, unsigned short sLen );
short EvWrite( unsigned char UserID, unsigned char DtIdx, unsigned char* pMsg, unsigned short sLen );
short CliEvWrite( unsigned char Client, unsigned char DtIdx, unsigned short DpIdx, unsigned char ItemIdx, unsigned char ItemLen, unsigned long Value );

/* fuer bksysgetinfo ----------- */
short GetDpInfo( char *pDpName, unsigned char *pDtIdx, unsigned short *pDpIdx, unsigned char **ppAlias );
short GetDtDescInfos( unsigned char DtIdx, DtProps_Typ **ppDtProps,
					  EaDesc_Typ **ppEaDesc, unsigned char *pEaDescMaxIdx,
					  DtDesc_Typ **ppDtDesc, unsigned char *pDtDescMaxIdx,
					  ItemConv_Typ **ppItemConv, unsigned char *pItemConvMaxIdx );

/* fuer bksysgetindex ---------- */
short GetItemIndex(DtDesc_Typ *pDtDesc, char *ItemName, short MaxItemIdx);
short GetDtIndex(DtProps_Typ *pProps, char *DtName, short MaxDtIdx);

/* fuer bksysgetpipe ----------- */
short EvGetPipePtr( unsigned char UserID, unsigned char DtIdx, PipeHead_Typ** ppPipe );
short CliGetPipePtr( unsigned char Client, unsigned char DtIdx, CliPipeHead_Typ** ppPipe );

/* fuer bksysinet -------------- */
void ErrStatisticsY( unsigned char *pErrMk, unsigned short ErrBit, unsigned short *pSyErr, unsigned char ErrStat1, unsigned char ErrStatN, unsigned short ErrNum, unsigned long ErrInfo, unsigned char *pErrPre, unsigned char *pErrText );
short EvRead( EvPbHead_Typ* pEvBlock, unsigned char DtIdx, unsigned char* pMsg, unsigned short sSize, unsigned short* pLen );
short EvInit( unsigned char UserID, unsigned short AnzEvPar[DT_ANZ], EvPbHead_Typ** ppEvBlockHead );
short EvCreate( unsigned char UserID, unsigned char DtIdx, unsigned short DpIdx, unsigned char EvTyp, unsigned char cLink, unsigned char cFlag );
short EvParaInit( unsigned char UserID, unsigned char DtIdx, unsigned short DpIdx, unsigned char *pItemName, short Hyst, short Intvl );
short EvLink( unsigned char UserID, unsigned char EvTyp, unsigned char DtIdx, unsigned short DpIdx);
short EvCheckLink( unsigned char UserID, unsigned char EvTyp, unsigned char DtIdx, unsigned short DpIdx);
short EvSetFlag( unsigned char UserID, unsigned char EvTyp, unsigned char DtIdx, unsigned short DpIdx);
short EvPbCreate( unsigned char UserID, EvPbHead_Typ** ppEvBlock, DtProps_Typ *pProps, EvPbHead_Typ** ppEvBlockHead );
char GetUserIndex( unsigned char UserID);
void EvPipeInit( PipeHead_Typ* pPipe, short sBufSize );

/* fuer bksysbrtcp ------------- */
void ClientDiagnose( void );

/* fuer BkTcp ---------- */
short CliGetClientAnzMax( unsigned char *pCliAnzMax );
short CliGetDtAnz( unsigned char *pDtAnz );
short CliItemLink( unsigned char Client, unsigned char DtIdx, unsigned short DpIdx, unsigned char ItemIdx, unsigned char Link );
short CliItemLinkAll( unsigned char Client, unsigned char Link );
short CliSetItemHyst( unsigned char Client, unsigned char DtIdx, unsigned short DpIdx, unsigned char ItemIdx, unsigned char Len, unsigned char *pHyst );
short CliForceWriteEvent( unsigned char DtIdx, unsigned short DpIdx, unsigned char ItemIdx );
short CliEvRead( unsigned char Client, unsigned char DtIdx, unsigned short *pDpIdx, unsigned char *pItemIdx, unsigned char *pItemLen, unsigned long *pValue );
short CliAktValToCabVal( DtProps_Typ *pDtProps, DtDesc_Typ *pDtDesc, unsigned char *pPab, CabItemEntry_Typ *pCab, unsigned char ItemIdx );

#endif /* BKSYS_H_ */
```

### bktcp.h
```c
/******************************************************************************
*    COPYRIGHT    BERNECKER + RAINER Industrie-Elektronik Ges.m.b.H           *
*******************************************************************************
*  Projekt:  Burklimat 2000
*  Teil:     Parser-Funktionen
*  Datei:    bktcp.h
*  Typ:      GNU-C (32 Bit)
*------------------------------------------------------------------------------
*  Revision: 01.00
*  Datum:    04-08-2003
*  Autor:    Martin Kurtz / MKrz
*------------------------------------------------------------------------------
*  Funktion: Globale Include-Datei.
*------------------------------------------------------------------------------
*  Rev.  | Datum    | Name | Kommentar
*  ------+----------+------+---------------------------------------------------
*  01.00 | 04-08-03 | MKrz | Datei-Erstellung
*        |          |      |
******************************************************************************/

/***********************************************************************/
/* Konstantendefinition                                                */
/***********************************************************************/

#define FALSE	0	/* logisch falsch */
#define TRUE	1	/* logisch wahr */

/* Parser-Zustände */
enum {	cCD_PARSER_STATE_COUNT,				/* Parser-Status: Zählen der Datenpunkte */
		cCD_PARSER_STATE_DEF,				/* Parser-Status: Anmelden der Datenpunkte */
		cCD_PARSER_STATE_READY,				/* Parser-Status: Fertig */
		cCD_PARSER_STATE_ERROR,
		cCD_PARSER_STATE_ERROR_READY	};	/* Parser-Status: Fehler */

#define	cSIZE_UNIT_FILTER					32

/* Default-Werte */
#define cTCP_DEFAULT_PORT					20001	/* Default Port */
#define cTCP_DEFAULT_TIMEOUT				60		/* Default Timeout */

#define cTCP_DEFAULT_UNIT					1		/* Default Anlage */
#define cTCP_DEFAULT_DEVICE					1		/* Default Gerät */

/* Bezeichner */
#define cKW_TCP_PORT			"Client"	/* Port */
#define cKW_TCP_PORT_NUMBER		"Port"		/* Port-Nummer */

#define cKW_TCP_TIMEOUT			"Client"	/* Timeout */
#define cKW_TCP_TIMEOUT_NUMBER	"Timeout"	/* Timeout-Wert */

#define cKW_TCP_UNIT			"Anlage"	/* Anlage */
#define cKW_TCP_UNIT_NUMBER		"Nr"		/* Anlagen-Nummer */

#define cKW_TCP_POINT			"Dp"		/* Datenpunkt */
#define	cKW_TCP_POINT_NUMBER	"Nr"		/* Datenpunkt-Nummer */

#define cKW_TCP_DM_FIRST		"tcppara"	/* Datenmodul-Name 1 */
#define cKW_TCP_DM_SECOND		"dplist"	/* Datenmodul-Name 2 */

#define	cKW_TCP_STATION			"UST"		/* Schlüsselwort für Station */
#define	cKW_TCP_SECTION			"TCP"		/* Schlüsselwort für Tcp-Section */

/* Fehler-Nummern */
#define	EC_MEM_ALLOC_NEED					0	/* Fehler bei Allokieren von Speicher */
#define	ET_MEM_ALLOC_NEED					"MEM="

#define	EC_TMP_ALLOC_NEED					1	/* Fehler bei Allokieren von Speicher */
#define	ET_TMP_ALLOC_NEED					"kB, TMP="

#define	EC_DPS_FOUND						2	/* Fehler bei Allokieren von Speicher */
#define	ET_DPS_FOUND						"gef.DP="

#define	EC_DPS_NOT_FOUND					3	/* Fehler bei Allokieren von Speicher */
#define	ET_DPS_NOT_FOUND					", n.gef.DP="

#define	EC_TCP_READY						4	/* Fehler bei Allokieren von Speicher */
#define	ET_TCP_READY						" bereit"

#define	EC_TCP_NOT_READY					5	/* Fehler bei Allokieren von Speicher */
#define	ET_TCP_NOT_READY					" nicht bereit"

#define	EC_DA_NOT_FOUND						6	/* Fehler bei Allokieren von Speicher */
#define	ET_DA_NOT_FOUND						"Datenmodul nicht vorhanden"

#define	EC_TMP_ALLOC						7	/* Fehler bei Allokieren von Speicher */
#define	ET_TMP_ALLOC						"Fehler bei Allokieren von Speicher"

#define	EC_DP_FOUND							8	/* Fehler bei Allokieren von Speicher */
#define	ET_DP_FOUND							":DP gefunden: "

#define	EC_DP_NOT_FOUND						9	/* Fehler bei Allokieren von Speicher */
#define	ET_DP_NOT_FOUND						":DP nicht gefunden:"

#define	EC_TCP_VERS							10	/* Fehler bei Allokieren von Speicher */
#define	ET_TCP_VERS							"V"

#define	EC_TCP_NOT_VERS						11	/* Fehler bei Allokieren von Speicher */
#define	ET_TCP_NOT_VERS						"B"

#define	EC_PARSER_READY						12	/* Fehler bei Allokieren von Speicher */
#define	ET_PARSER_READY						":Parser bereit"

#define	EC_PARSER_STATE						13	/* Fehler im Parser-Zustand */
#define	ET_PARSER_STATE						":Syntax-Fehler -"

#define	EC_PARSER_STATIONTYPPOINT			14	/* Fehler im Parser-Zustand: Station/Typ/Punkt */
#define	ET_PARSER_STATIONTYPPOINT			":DP-Attr unbekannt"

#define	EC_PARSER_SECTION					15	/* Fehler im Parser-Zustand: Section */
#define	ET_PARSER_SECTION					":DP-Attr unbekannt"

#define	EC_PARSER_DATA						16	/* Fehler im Parser-Zustand: Data */
#define	ET_PARSER_DATA						":DP-Attr unbekannt"

#define	EC_NO_PGLOBALS						17	/* Fehler, da kein gültiger pGlobals-Pointer */
#define	ET_NO_PGLOBALS						":kein pGlobals"

#define	EC_PORT_ALREADY_EXISTS				18	/* Fehler, da Port bereits vergeben */
#define	ET_PORT_ALREADY_EXISTS				":Port bereits vorh."

#define	EC_TIMEOUT_ALREADY_EXISTS			19	/* Fehler, da Tiemout bereits vergeben */
#define	ET_TIMEOUT_ALREADY_EXISTS			":Timeout bereits vorh"

#define	EC_POINT_ALREADY_EXISTS				20	/* Fehler, da Datenpunkt bereits existiert */
#define	ET_POINT_ALREADY_EXISTS				":Dp bereits vorhanden"

#define	EC_MAX								21	/* Anzahl Fehlereinträge */

/***********************************************************************/
/* Datentypdeklaration                                                 */
/***********************************************************************/

typedef plcbit BIT;			/* Datentyp BIT */

/* ---------------------------------- */
/* Datentypen für Zugriff von Tcp aus */
/* ---------------------------------- */
typedef struct {
	long					TcpPoint;
	unsigned short			Bk2Point;
	unsigned char			*pAlias;
} TCP_ACCESS_BK2_POINT;

typedef struct {
	unsigned short			countTcpPoints;
	TCP_ACCESS_BK2_POINT	*pTcpAccessBk2Point;
} TCP_ACCESS_BK2_TYPE;

typedef struct {
	long					TcpUnit;
	unsigned long			countTcpUnitPoints;
	TCP_ACCESS_BK2_TYPE		*pTcpAccessBk2Type;
} TCP_ACCESS_BK2_UNIT;

typedef struct {
	unsigned short			countTcpUnits;
	TCP_ACCESS_BK2_UNIT		*pTcpAccessBk2Unit;
} TCP_ACCESS_BK2_SYSTEM;

/* ---------------------------------- */
/* Datentypen für Zugriff von Bk2 aus */
/* ---------------------------------- */
typedef struct {
	long					TcpUnit;
	long					TcpPoint;
	unsigned char			*pAlias;
} BK2_ACCESS_TCP_POINT;

typedef struct {
	unsigned short			countBk2Points;
	BK2_ACCESS_TCP_POINT	*pBk2AccessTcpPoint;
} BK2_ACCESS_TCP_TYPE;

typedef struct {
	unsigned short			countBk2Types;
	BK2_ACCESS_TCP_TYPE		*pBk2AccessTcpType;
} BK2_ACCESS_TCP_SYSTEM;

/***********************************************************************/
/* inetbk2-Funktionen                                                  */
/***********************************************************************/
unsigned char IsANumber(unsigned char *pData);
int ltoa(long value, char *buffer);
int ultoa(unsigned long value, char *buffer);

/*============================= Ende der Datei ==============================*/
```

### brtcp.h
```c
/* TCP/IP definitions > configuration data ! */
#define MAX_CLIENTS	8
#define MYADRS	ETH_INADDR_ANY
#define RECVBUFLEN		1024
#define SENDBUFLEN		2048

#define FALSE		0
#define TRUE		1
#define NULL 		0

/* AK-codes */
#define BRT_ITM_LOGON			1
#define BRT_ITM_LOGON_TS		2
#define BRT_ITM_LOGOFF			3
#define BRT_ITM_READ			4
#define BRT_ITM_READ_TS			5
#define BRT_ITM_WRITE			6
#define BRT_ITM_EVENT			7
#define BRT_ITM_EVENT_TS		8
#define BRT_DATASTREAM_READ		9
#define BRT_CLI_WATCHDOG		10
#define BRT_TIMESYNC			11
#define BRT_DATASTREAM			12

#define BRT_ITM_LOGON_OK		101
#define BRT_ITM_LOGON_TS_OK		102
#define BRT_ITM_LOGOFF_OK		103
#define BRT_ITM_READ_OK			104
#define BRT_ITM_READ_TS_OK		105
#define BRT_ITM_WRITE_OK		106
#define BRT_DATASTREAM_READ_OK	109
#define BRT_CLI_WATCHDOG_OK		110
#define BRT_TIMESYNC_OK			111

#define BRT_CLI_ERROR			200
#define BRT_ITM_LOGON_ERR		201
#define BRT_ITM_LOGOFF_ERR		203
#define BRT_ITM_READ_ERR		204
#define BRT_ITM_WRITE_ERR		206
#define BRT_DATASTREAM_READ_ERR	209
#define BRT_TIMESYNC_ERR		211

/* error codes */
#define BRT_ERR_INVALIDAK			1
#define BRT_ERR_NO_ITEM				2
#define BRT_ERR_WRONG_LEN			3
#define BRT_ERR_WRONG_HYST			4
#define BRT_ERR_IS_LOGGED			5
#define BRT_ERR_ITEM_NO_TS			6

#define BRT_ERR_ITEM_NO_LOGON		7

#define BRT_ERR_NO_STREAM			8

#define BRT_ERR_RTC_SET				9

#define BRT_ERR_ITEM_NOT_WRITEABLE	10
#define BRT_ERR_WRITE_PIPE_FULL		11
#define BRT_ERR_ITEM_NO_DATA		12
#define BRT_ERR_SWC_SET				13

#define BRT_ERR_UNKNOWN_UNIT		14
#define BRT_ERR_UNKNOWN_DEVICE		15
#define BRT_ERR_UNKNOWN_TYPE		16
#define BRT_ERR_UNKNOWN_POINT		17
#define BRT_ERR_WRONG_ITEM			18

enum {CLI_INIT, CLI_CONNECTED, CLI_DISCONNECTED, CLI_ERROR, CLI_WATCHDOG, CLI_SENDERROR, CLI_STATUSANZAHL };	/* für client-Status */
enum {STREAM_IDLE, STREAM_INIT, STREAM_BUSY, STREAM_READY};

typedef struct{
	DINT				socket;
	INT					status;
	ETH_sockaddr_typ	client_str;
	UINT				recv_cnt;
	TON_typ				TON_watchdog;
	UDINT				recv_in;
	UDINT				recv_out;
	UDINT				send_in;
	UDINT				send_out;
	USINT				recv_buf[RECVBUFLEN];
	USINT				send_buf[SENDBUFLEN];
	UINT				EventID;
	UINT				startType;
	INT					stateEvRead;
	USINT				EventBuffer[256];
	UDINT				lenEventMessage;
	UDINT				lengthTimeStamp;
	UINT				EventCnt;
	UINT				stateStream;
	USINT				*pStreamData;
	INT					stateRelease;
} client_typ;

typedef struct {
	UINT				ID;
	UINT				AK;
} CLI_HEAD_TYP;

typedef struct {
	UINT				anlage;
	UINT				geraet;
	UINT				typ;
	UINT				punkt;
	UINT				item;
} CLI_ADR_TYP;

typedef struct {
	CLI_HEAD_TYP		head;
	CLI_ADR_TYP			Adr;
	UINT				LenLow;
	UINT				LenHigh;
	UINT				Data;
} CLI_LOGON_REQUEST;

typedef struct {
	CLI_HEAD_TYP		head;
	CLI_ADR_TYP			Adr;
	UINT				LenLow;
	UINT				LenHigh;
	UINT				Data;
} CLI_LOGON_RESPONSE;

typedef struct {
	CLI_HEAD_TYP		head;
	CLI_ADR_TYP			Adr;
} CLI_LOGOFF_REQUEST;

typedef struct {
	CLI_HEAD_TYP		head;
	CLI_ADR_TYP			Adr;
} CLI_LOGOFF_RESPONSE;

typedef struct {
	CLI_HEAD_TYP		head;
	CLI_ADR_TYP			Adr;
} CLI_READ_REQUEST;

typedef struct {
	CLI_HEAD_TYP		head;
	CLI_ADR_TYP			Adr;
	UINT				LenLow;
	UINT				LenHigh;
	UINT				Data;
} CLI_READ_RESPONSE;

typedef struct {
	CLI_HEAD_TYP		head;
	CLI_ADR_TYP			Adr;
	UINT				LenLow;
	UINT				LenHigh;
	UINT				Data;
} CLI_WRITE_REQUEST;

typedef struct {
	CLI_HEAD_TYP		head;
	CLI_ADR_TYP			Adr;
} CLI_WRITE_RESPONSE;

typedef struct {
	CLI_HEAD_TYP		head;
	CLI_ADR_TYP			Adr;
	UINT				LenLow;
	UINT				LenHigh;
	UINT				Data;
} CLI_EVENT_RESPONSE;

typedef struct {
	CLI_HEAD_TYP		head;
	UINT				Error;
} CLI_ERROR_RESPONSE;

typedef struct {
	CLI_HEAD_TYP		head;
	CLI_ADR_TYP			Adr;
	UINT				Error;
} CLI_ADRERROR_RESPONSE;

typedef struct {
	CLI_HEAD_TYP		head;
} CLI_WATCHDOG_REQUEST;

typedef struct {
	CLI_HEAD_TYP		head;
} CLI_WATCHDOG_RESPONSE;

typedef struct {
	CLI_HEAD_TYP		head;
	RTCtime_typ			Time;
} CLI_TIMESYNC_REQUEST;

typedef struct {
	CLI_HEAD_TYP		head;
} CLI_TIMESYNC_RESPONSE;

typedef struct {
	CLI_HEAD_TYP		head;
	CLI_ADR_TYP			Adr;
	UINT				LenLow;
	UINT				LenHigh;
} CLI_DATASTREAM;
```

### bsrun.h
```c
/******************************************************************************
*    COPYRIGHT    BERNECKER + RAINER Industrie-Elektronik Ges.m.b.H           *
*******************************************************************************
*  Projekt:  BrServer
*  Teil:     Header-File
*  Datei:    bsrun.h
*  Typ:      GNU C (32 Bit)
*------------------------------------------------------------------------------
*  Revision: 01.00
*  Datum:    04-08-2003
*  Autor:    Martin Kurtz / MKrz
*------------------------------------------------------------------------------
*  Funktion: Generelle Definitionen.
*------------------------------------------------------------------------------
*  Rev.  | Datum    | Name | Kommentar
*  ------+----------+------+---------------------------------------------------
*  01.00 | 14-07-03 | MKrz | Datei-Erstellung
*        |          |      |
******************************************************************************/

/* --------------------- */
/* logische Definitionen */
/* --------------------- */
#define FALSE	0
#define TRUE	1

/* ---------------------------- */
/* Zustände für Initialisierung */
/* ---------------------------- */
#define cSTATE_INIT_COUNT		0
#define cSTATE_INIT_ALLOC		1
#define cSTATE_INIT_READY		2

/* ------------------- */
/* Fehler-Definitionen */
/* ------------------- */
#define cEC_OK						0

#define cEC_INVALID_SERVER			1000
#define cEC_INVALID_INSTANCE		1001
#define cEC_INVALID_UNIT			1002
#define cEC_INVALID_DEVICE			1003
#define cEC_INVALID_TYPE			1004
#define cEC_INVALID_POINT			1005
#define cEC_INVALID_ITEM			1006
#define cEC_INVALID_VALUE			1007

#define cEC_INVALID_TYPE_FOR_HYST	1100
#define cEC_INVALID_POINT_FOR_HYST	1101

#define cEC_NO_DATA_IN_EVENTBUFFER	1200
#define cEC_EVENTBUFFER_TO_SMALL	1201
#define cEC_INVALID_LENGTH_IN_EVENT	1202

#define cEC_ITEM_ALREADY_LINKED		1300
#define cEC_ITEM_ALREADY_UNLINKED	1301
#define cEC_ITEM_NO_TIMESTAMP		1302

#define cEC_INVALID_LENGTH			1400
#define cEC_INVALID_HANDLE			1401

#define cEC_ITEM_NOT_WRITEABLE		1500
#define cEC_NO_DATA_IN_WRITEBUFFER	1501
#define cEC_WRITE_PIPE_FULL			1502

/* ------------------- */
/* Status-Definitionen */
/* ------------------- */
enum {	cITEM_UNLINKED,
		cITEM_LINKED_WITHOUT_TIMESTAMP,
		cITEM_LINKED_WITH_TIMESTAMP	};

#define cMAX_INSTANCE	16

/* ------------------------------ */
/* Datentypen für Initialisierung */
/* ------------------------------ */
typedef struct {
	UINT	word_0;
	UINT	word_1;
} UNIT_DEFINITION;

typedef struct {
	UINT	word_0;
	UINT	word_1;
} DEVICE_DEFINITION;

typedef struct {
	USINT	length_extern;
	USINT	signed_extern;
	USINT	length_intern;
	USINT	signed_intern;
	USINT	time_stamp;
	USINT	hyst;
	USINT	typeforhyst;
	USINT	init;
	UINT	init_value;
	UINT	pipe_entry;
} TYPE_DEFINITION;

/* ------------------------- */
/* Datentypen für Eventpipes */
/* ------------------------- */
typedef struct {
	UDINT	countEvent;
	UDINT	firstEvent;
	UDINT	lastEvent;
} PIPE_EVENT_STATE;

typedef struct {
	PIPE_EVENT_STATE	stateEvent;
	UINT	pipe_entry;
	UINT	pipe_size;
	UINT	pipe_level;
	USINT*	pPipeData;
	UINT	iPipeRead;
	UINT	iPipeWrite;
} EVENT_PIPE_HEADER;

typedef struct {
	USINT	linkstate;
	USINT	eventtype;
	UINT	unit;
	UINT	device;
	UINT	type;
	UINT	point;
	UINT	item;
	UDINT	length;
	USINT*	pData;
} EVENT_PIPE_DATA;

typedef struct {
	EVENT_PIPE_HEADER*	pEventPipeHeader;
	UDINT				length_pipe_next;
	TYPE_DEFINITION		TypeDefinition;
} ACCESS_EVENT_PIPE;

typedef struct {
	UINT	pipe_entry;
	UINT	pipe_size;
	UINT	pipe_level;
	USINT*	pPipeData;
	UINT	iPipeRead;
	UINT	iPipeWrite;
} WRITE_PIPE_HEADER;

typedef struct {
	USINT	linkstate;
	USINT	eventtype;
	UINT	unit;
	UINT	device;
	UINT	type;
	UINT	point;
	UINT	item;
	UDINT	length;
	USINT*	pData;
} WRITE_PIPE_DATA;

typedef struct {
	WRITE_PIPE_HEADER*	pWritePipeHeader;
	UDINT				length_pipe_next;
} ACCESS_WRITE_PIPE;

/* ---------------------------------------- */
/* Datentypen für Zugriff auf Prozessabbild */
/* ---------------------------------------- */
typedef USINT	ACCESS_ITEM_VALID;
typedef	USINT	ACCESS_ITEM_EVENT_LINK;

typedef USINT	POINT_LINK_STATE;
typedef USINT	POINT_VALID_STATE;
typedef USINT	POINT_RELEASE_STATE;

typedef	UINT	ACCESS_ITEM_WRITE_LINK;
typedef	UDINT	ACCESS_ITEM_WRITE_HANDLE;

typedef struct {
	UDINT	noEvent;
} POINT_EVENT_STATE;

typedef struct {
	UDINT	countEvent;
} TYPE_EVENT_STATE;

typedef struct {
	UDINT	countEvent;
} DEVICE_EVENT_STATE;

typedef struct {
	UDINT	countEvent;
} UNIT_EVENT_STATE;

typedef struct {
	UDINT	countEvent;
} SERVER_EVENT_STATE;

typedef struct {
	UINT	countPoint;

	USINT*	pData_extern;
	UINT	length_extern;
	UINT	length_extern_align;

	USINT*	pData_intern;
	UINT	length_intern;
	UINT	length_intern_align;

	USINT*	pData_iextern;
	UINT	length_iextern;
	UINT	length_iextern_align;
	UINT	length_iextern_next;

	USINT*	pData_valid;
	UINT	length_valid;
	UINT	length_valid_align;

	USINT*	pData_time;
	UINT	length_time;
	UINT	length_time_align;

	USINT*	pData_itime;
	UINT	length_itime;
	UINT	length_itime_align;
	UINT	length_itime_next;

	USINT*	pData_writelink;
	UINT	length_writelink;
	UINT	length_writelink_align;

	USINT*	pData_writehandle;
	UINT	length_writehandle;
	UINT	length_writehandle_align;

	USINT*	pData_ieventlink;
	UINT	length_ieventlink;
	UINT	length_ieventlink_align;
	UINT	length_ieventlink_next;

	USINT*	pData_ireleasestream;
	UINT	length_ireleasestream;
	UINT	length_ireleasestream_align;
	UINT	length_ireleasestream_next;

	USINT*	pData_ihyst;
	UINT	length_ihyst;
	UINT	length_ihyst_align;
	UINT	length_ihyst_next;

	USINT*	pData_ievent;
	UINT	length_ievent;
	UINT	length_ievent_align;
	UINT	length_ievent_next;
} ACCESS_TYPE;

typedef struct {
	UINT				countType;
	UINT				device_no;
	ACCESS_TYPE*		pAccessType;
	TYPE_EVENT_STATE*	pTypeEventState;
} ACCESS_DEVICE;

typedef struct {
	UINT				countDeviceNo;
	UINT				unit_no;
	ACCESS_DEVICE*		pAccessDevice;
	DEVICE_EVENT_STATE*	pDeviceEventState;
} ACCESS_UNIT;

typedef struct {
	UINT				countEventInstance;
	UINT				countWriteInstance;
	UINT				countType;
	UINT				countUnitNo;
	ACCESS_UNIT*		pAccessUnit;
	UNIT_EVENT_STATE*	pUnitEventState;
	ACCESS_EVENT_PIPE*	pAccessEventPipe;
	ACCESS_WRITE_PIPE*	pAccessWritePipe;
	UINT				PortNumber;
	UINT				TimeoutValue;
} ACCESS_SERVER;

/* ----------------------- */
/* Funktionen für Brserver */
/* ----------------------- */
UINT GetIdBrServer (void **pidBrServer, UINT *pbrstate);
UINT GetPortNumber (void *idBrServer, UINT *pPortNumber);
UINT GetTimeoutValue (void *idBrServer, UINT *pTimeoutValue);
UINT GetEventInstanceInfo (void *idBrServer, UINT *pEventInstance);
UINT GetWriteInstanceInfo (void *idBrServer, UINT *pWriteInstance);
UINT GetTypeInfo (void *idBrServer, UINT *ptype);
UINT GetItemInfo (void *idBrServer, UINT instance,
					UINT unit, UINT device, UINT type, UINT point, UINT item,
					USINT** ppData_extern,		UDINT* plength_extern,
					USINT** ppData_intern,		UDINT* plength_intern,
					USINT** ppData_iextern,		UDINT* plength_iextern,
					USINT** ppData_valid,		UDINT* plength_valid,
					USINT** ppData_time,		UDINT* plength_time,
					USINT** ppData_itime,		UDINT* plength_itime,
					USINT** ppData_writelink,	UDINT* plength_writelink,
					USINT** ppData_ieventlink,	UDINT* plength_ieventlink,
					USINT** ppData_ihyst,		UDINT* plength_ihyst,
					USINT** ppData_ievent,		UDINT* plength_ievent);
UINT GetEventLinkInfo (void *idBrServer,
						UINT unit, UINT device, UINT type, UINT point, UINT item,
						UINT *pcountInstanceAll, UINT *pcountInstanceNoTimestamp, UINT *pcountInstanceTimestamp);
UINT GetEventPipeInfo (void *idBrServer, UINT instance, UINT type,
						UINT *pipe_entry, UINT *pipe_level_abs, USINT *pipe_level_rel);
UINT GetWritePipeInfo (void *idBrServer, UINT instance,
						UINT *pipe_entry, UINT *pipe_level_abs, USINT *pipe_level_rel);
UINT LinkEventInstance (void *idBrServer, UINT instance);
UINT UnlinkEventInstance (void *idBrServer, UINT instance);
UINT LinkEventUnit (void *idBrServer, UINT instance,
					UINT unit);
UINT UnLinkEventUnit (void *idBrServer, UINT instance,
						UINT unit);
UINT LinkEventDevice (void *idBrServer, UINT instance,
						UINT unit, UINT device);
UINT UnLinkEventDevice (void *idBrServer, UINT instance,
						UINT unit, UINT device);
UINT LinkEventType (void *idBrServer, UINT instance,
					UINT unit, UINT device, UINT type);
UINT UnlinkEventType (void *idBrServer, UINT instance,
						UINT unit, UINT device, UINT type);
UINT LinkEventItem (void *idBrServer, UINT instance,
					UINT unit, UINT device, UINT type, UINT point, UINT item,
					USINT timestamp);
UINT UnlinkEventItem (void *idBrServer, UINT instance,
						UINT unit, UINT device, UINT type, UINT point, UINT item);
UINT SetHystItem (void *idBrServer, UINT instance,
					UINT unit, UINT device, UINT type, UINT point, UINT item,
					USINT* pValue, UDINT lengthValue);
UINT SetValueItem (void *idBrServer,
					UINT unit, UINT device, UINT type, UINT point, UINT item,
					USINT* pValue, UDINT lengthValue,
					RTCtime_typ RTCTime, USINT setTimeStampNow,
					USINT enableEvent);
UINT GetValueItem (void *idBrServer, UINT instance,
					UINT unit, UINT device, UINT type, UINT point, UINT item,
					USINT** ppData_extern, UDINT* plength_extern,
					USINT** ppData_time, UDINT* plength_time);
UINT SetEventItem (void *idBrServer, UINT instance,
					UINT unit, UINT device, UINT type, UINT point, UINT item,
					USINT* pValue, UINT lengthValue,
					USINT eventtype, USINT* pDataExtern, RTCtime_typ RTCTime);
UINT SetEventItemStream (void *idBrServer,
							UINT unit, UINT device, UINT type, UINT point, UINT item,
							USINT* pValue, UDINT lengthValue,
							USINT* pFlag,
							RTCtime_typ RTCTime, USINT setTimeStampNow,
							USINT enableEvent);
UINT ReleaseEventItemStream (void *idBrServer, UINT instance,
								UINT unit, UINT device, UINT type, UINT point, UINT item);
UINT GetEventItem (void *idBrServer, UINT instance,
					UINT type, USINT* pEventBuffer, UDINT lengthEventBuffer,
					UDINT* pLength, UDINT* pLengthTimeStamp);
UINT WorkEvent (void *idBrServer);
UINT LinkWriteInstance (void *idBrServer, UINT instance);
UINT UnlinkWriteInstance (void *idBrServer, UINT instance);
UINT LinkWriteUnit (void *idBrServer, UINT instance,
					UINT unit);
UINT UnlinkWriteUnit (void *idBrServer, UINT instance,
						UINT unit);
UINT LinkWriteDevice (void *idBrServer, UINT instance,
						UINT unit, UINT device);
UINT UnlinkWriteDevice (void *idBrServer, UINT instance,
						UINT unit, UINT device);
UINT LinkWriteType (void *idBrServer, UINT instance,
					UINT unit, UINT device, UINT type);
UINT UnlinkWriteType (void *idBrServer, UINT instance,
						UINT unit, UINT device, UINT type);
UINT LinkWriteItem (void *idBrServer, UINT instance,
					UINT unit, UINT device, UINT type, UINT point, UINT item,
					UDINT handle);
UINT UnlinkWriteItem (void *idBrServer, UINT instance,
						UINT unit, UINT device, UINT type, UINT point, UINT item);
UINT SetWriteItem (void *dBrServer,
					UINT unit, UINT device, UINT type, UINT point, UINT item,
					USINT* pValue, UDINT lengthValue);
UINT GetWriteItem (void *idBrServer, UINT instance,
					USINT* pWriteBuffer, UDINT lengthWriteBuffer,
					UDINT* pLength, UDINT* pLengthTimeStamp);

/*============================= Ende der Datei ==============================*/
```

### dbserv.h
```c
/******************************************************************************
*    COPYRIGHT    BERNECKER + RAINER Industrie-Elektronik Ges.m.b.H           *
*******************************************************************************
*  Projekt:  DbServ
*  Teil:     Parser-Funktionen
*  Datei:    dbserv.h
*  Typ:      GNU-C (32 Bit)
*------------------------------------------------------------------------------
*  Revision: 01.03
*  Datum:    04-08-2003
*  Autor:    Martin Kurtz / MKrz
*------------------------------------------------------------------------------
*  Funktion: Globale Include-Datei.
*------------------------------------------------------------------------------
*  Rev.  | Datum    | Name | Kommentar
*  ------+----------+------+---------------------------------------------------
*  01.03 | 26-07-04 | MKrz | Typzuordnung verbessert
*  01.01 | 06-07-04 | MKrz | Fehlermeldungen angepasst
*  01.00 | 04-08-03 | MKrz | Datei-Erstellung
*        |          |      |
******************************************************************************/

/***********************************************************************/
/* Konstantendefinition                                                */
/***********************************************************************/

#define FALSE	0	/* logisch falsch */
#define TRUE	1	/* logisch wahr */

#ifndef ERR_FUB_BUSY
	#define ERR_FUB_BUSY	0xFFFF
#endif

/* Instanznummern Schreiben */
enum {	cINSTANCE_DBSLIB,
		cINSTANCE_IODRV,
		cINSTANCE_IEC103,
		cINSTANCE_L2DP	};

/* Parser-Zustände */
enum {	cCD_PARSER_STATE_DEF_TCP,			/* Parser-Zustand  0: Tcp-Definitionen */

		cCD_PARSER_STATE_DEF_BUF,			/* Parser-Zustand  1: Buf-Definitionen */

		cCD_PARSER_STATE_COUNT_TYPE,		/* Parser-Zustand  2: Zählen der Datentypen */
		cCD_PARSER_STATE_DEF_TYPE,			/* Parser-Zustand  3: Anmelden der Datentypen */

		cCD_PARSER_STATE_COMPARE_DO_TYPE,	/* Parser-Zustand  4: Abgleich der Datentypdefinitionen */
		cCD_PARSER_STATE_DEL_DO_TYPE,		/* Parser-Zustand  5: Löschen des Datenobjektes für Datentypdefinitionen */
		cCD_PARSER_STATE_CREATE_DO_TYPE,	/* Parser-Zustand  6: Anlegen des Datenobjektes für Datentypdefinitionen */

		cCD_PARSER_STATE_COUNT_DP,			/* Parser-Zustand  7: Zählen der Datenpunkte */
		cCD_PARSER_STATE_DEF_DP,			/* Parser-Zustand  8: Anmelden der Datenpunkte */

		cCD_PARSER_STATE_COMPARE_DO_POINT,	/* Parser-Zustand  9: Abgleich der Datentypdefinitionen */
		cCD_PARSER_STATE_DEL_DO_POINT,		/* Parser-Zustand 10: Löschen des Datenobjektes für Datentypdefinitionen */
		cCD_PARSER_STATE_CREATE_DO_POINT,	/* Parser-Zustand 11: Anlegen des Datenobjektes für Datentypdefinitionen */

		cCD_PARSER_STATE_ALLOC_ACCESS_DATA,	/* Parser-Zustand 12: Prozessabbild allokieren */

		cCD_PARSER_STATE_COMPARE_DO_DATA,	/* Parser-Zustand 13: Abgleich der Datentypdefinitionen */
		cCD_PARSER_STATE_DEL_DO_DATA,		/* Parser-Zustand 14: Löschen des Datenobjektes für Datentypdefinitionen */
		cCD_PARSER_STATE_CREATE_DO_DATA,	/* Parser-Zustand 15: Anlegen des Datenobjektes für Datentypdefinitionen */

		cCD_PARSER_STATE_WORK_DATA,			/* Parser-Zustand 16: */

		cCD_PARSER_STATE_COMPARE_DO_EVENT,	/* Parser-Zustand 17: Abgleich der Datentypdefinitionen */
		cCD_PARSER_STATE_DEL_DO_EVENT,		/* Parser-Zustand 18: Löschen des Datenobjektes für Datentypdefinitionen */
		cCD_PARSER_STATE_CREATE_DO_EVENT,	/* Parser-Zustand 19: Anlegen des Datenobjektes für Datentypdefinitionen */

		cCD_PARSER_STATE_GET_DEVMEMINFO,	/* Parser-Zustand 20: */
		cCD_PARSER_STATE_WORK_EVENT,		/* Parser-Zustand 21: */

		cCD_PARSER_STATE_READY,				/* Parser-Zustand 22: Fertig */
		cCD_PARSER_STATE_ERROR,				/* Parser-Zustand 23: Fehler */
		cCD_PARSER_STATE_ERROR_READY	};	/* Parser-Zustand 24: Fertig mit Fehler */

/* Default-Werte */
#define cTCP_DEFAULT_PORT			20001		/* Default Port */
#define cTCP_DEFAULT_TIMEOUT		20			/* Default Timeout */

#define cDBS_DEFAULT_UNIT			1			/* Default Anlage */
#define cDBS_DEFAULT_DEVICE			1			/* Default Gerät */

/* Max-Werte */
#define cMAX_UNIT_DEF				65535		/* maximaler Wert */
#define cMAX_TYPE_DEF				65535		/* maximaler Wert */
#define cMAX_POINT_DEF				65535		/* maximaler Wert */

/* Bezeichner */
#define cKW_DBS_DM_DP_LIST			"dplist"	/* Datenmodul-Name 1 */
#define cKW_DBS_DM_TYP_LIST			"typlist"	/* Datenmodul-Name 2 */

#define cKW_ITEM_SECTION			"ITEM"		/* Schlüsselwort für Item-Section */
#define cKW_ALL_SECTION				"ALL"		/* Schlüsselwort für All-Section */
#define cKW_DBS_SECTION				"DBS"		/* Schlüsselwort für Dbs-Section */

#define cKW_BUF_SECTION				"BUF"		/* Schlüsselwort für Buf-Section */

#define cKW_DBS_CLIENT				"Client"	/* Instanzen */
#define cKW_DBS_CLIENT_COUNT		"Anz"		/* Instanzen-Anzahl */
#define cKW_DBS_APP					"App"		/* Applikation */
#define cKW_DBS_APP_COUNT			"Anz"		/* Applikation-Anzahl */
#define cKW_DBS_UNIT				"Anlage"	/* Anlage */
#define cKW_DBS_UNIT_NUMBER			"Nr"		/* Anlagen-Nummer */
#define cKW_DBS_TYPE				"Typ"		/* Datentyp */
#define cKW_DBS_TYPE_NUMBER			"Nr"		/* Datentyp-Nummer */

#define cKW_DBS_TYPE_FILE_SIZE		"FbSize"	/* Datentyp-Filebuffer Grösse */
#define cKW_DBS_TYPE_FILE_MODE		"FbMode"	/* Datentyp-Filebuffer Modus */

#define cKW_DBS_BUF_ATTRIBUTE		"Buf"		/* Datentyp-Filebuffer Modus */
#define cKW_DBS_BUF_EVENTS			"Events"	/* Datentyp-Filebuffer Modus */
#define cKW_DBS_BUF_TYPE			"Typ"		/* Datentyp-Filebuffer Modus */

#define cKW_DBS_ITEM				"Item"		/* Datentyp-Item */
#define cKW_DBS_ITEM_NUMBER			"Nr"		/* Datentyp-Item-Nummer */
#define cKW_DBS_ITEM_NAME			"Name"		/* Datentyp-Item-Name */
#define cKW_DBS_TYPE_TIMESTAMP		"TS"		/* Datentypbezeichner für Zeitstempel */
#define cKW_DBS_POINT				"Dp"		/* Datenpunkt */
#define cKW_DBS_POINT_NUMBER		"Nr"		/* Datenpunkt-Nummer */
#define cKW_DBS_FUB					"Fub"		/* Funktionsblock */

#define cKW_DBS_TYPE_BOOL			"_BOOL"		/* Datentypbezeichner für BOOL */
#define cKW_DBS_TYPE_USINT			"_USINT"	/* Datentypbezeichner für USINT */
#define cKW_DBS_TYPE_SINT			"_SINT"		/* Datentypbezeichner für SINT */
#define cKW_DBS_TYPE_UINT			"_UINT"		/* Datentypbezeichner für UINT */
#define cKW_DBS_TYPE_INT			"_INT"		/* Datentypbezeichner für INT */
#define cKW_DBS_TYPE_UDINT			"_UDINT"	/* Datentypbezeichner für UDINT */
#define cKW_DBS_TYPE_DINT			"_DINT"		/* Datentypbezeichner für DINT */
#define cKW_DBS_TYPE_STREAM			"_STREAM"	/* Datentypbezeichner für STREAM */

/* Typ-IDs */
enum {	cDBS_IDTYPE_UNDEF,
		cDBS_IDTYPE_BOOL,
		cDBS_IDTYPE_USINT,
		cDBS_IDTYPE_SINT,
		cDBS_IDTYPE_UINT,
		cDBS_IDTYPE_INT,
		cDBS_IDTYPE_UDINT,
		cDBS_IDTYPE_DINT,
		cDBS_IDTYPE_STREAM	};

/* Typ-Eigenschaften */
enum {	cDBS_TYPE_UNSIGNED,					/* vorzeichenloser Typ */
		cDBS_TYPE_SIGNED,					/* vorzeichenbehafteter Typ */
		cDBS_TYPE_STREAM	};				/* Zeiger auf Datenstrom */

/* Bezeichner */
#define cKW_TCP_PORT			"Client"	/* Port */
#define cKW_TCP_PORT_NUMBER		"Port"		/* Port-Nummer */

#define cKW_TCP_TIMEOUT			"Client"	/* Timeout */
#define cKW_TCP_TIMEOUT_NUMBER	"Timeout"	/* Timeout-Wert */

#define cKW_TCP_STATION			"UST"		/* Schlüsselwort für Station */
#define cKW_TCP_SECTION			"TCP"		/* Schlüsselwort für Station */

/* Fehler-Nummern */
#define EC_MEM_ALLOC_NEED			0	/* Benötigter Mem-Speicher */
#define ET_MEM_ALLOC_NEED			"MEM="

#define EC_TMP_ALLOC_NEED			1	/* Benötigter Tmp-Speicher */
#define ET_TMP_ALLOC_NEED			"kB, TMP="

#define EC_DPS_FOUND				2	/* gefundene Datenpunkte */
#define ET_DPS_FOUND				"gef.DP="

#define EC_DPS_NOT_FOUND			3	/* nicht gefundene Datenpunkte */
#define ET_DPS_NOT_FOUND			", n.gef.DP="

#define EC_ITEM_NOT_FOUND			4	/* nicht gefundenes Item */
#define ET_ITEM_NOT_FOUND			", n.gef.ITEM="

#define EC_ITEM_INVALID_FOUND		5	/* nicht gefundenes Item */
#define ET_ITEM_INVALID_FOUND		"unerw.gef.ITEM="

#define EC_TCP_READY				6	/* TCP bereit */
#define ET_TCP_READY				" bereit"

#define EC_TCP_NOT_READY			7	/* TCP nicht bereit */
#define ET_TCP_NOT_READY			" nicht bereit"

#define EC_DA_NOT_FOUND				8	/* Datenmodul nicht gefunden */
#define ET_DA_NOT_FOUND				"Datenmodul nicht vorhanden"

#define EC_TMP_ALLOC				9	/* Fehler bei Allokieren von Speicher */
#define ET_TMP_ALLOC				"Fehler bei Allokieren von Speicher"

#define EC_ITEM_NO_INVALID			10	/* Item-Nummer falsch */
#define ET_ITEM_NO_INVALID			":ITEM Nr falsch: "

#define EC_ITEM_ALREADY_EXIST		11	/* Item-Name falsch */
#define ET_ITEM_ALREADY_EXIST		":ITEM Name falsch: "

#define EC_DP_FOUND					12	/* Datenpunkt gefunden */
#define ET_DP_FOUND					":DP gefunden: "

#define EC_DP_NOT_FOUND				13	/* Datenpunkt nicht gefunden */
#define ET_DP_NOT_FOUND				":DP nicht gefunden:"

#define EC_TCP_VERS					14	/* Zeichen für Vollversion */
#define ET_TCP_VERS					"V"

#define EC_TCP_NOT_VERS				15	/* Zeichen für Vorabversion */
#define ET_TCP_NOT_VERS				"B"

#define EC_PARSER_READY				16	/* Parser bereit */
#define ET_PARSER_READY				":Parser bereit"

#define EC_PARSER_STATE				17	/* Fehler im Parser-Zustand */
#define ET_PARSER_STATE				":Syntax-Fehler -"

#define EC_PARSER_STATIONTYPPOINT	18	/* Fehler im Parser-Zustand: Station/Typ/Punkt */
#define ET_PARSER_STATIONTYPPOINT	":DP-Attr unbekannt"

#define EC_PARSER_SECTION			19	/* Fehler im Parser-Zustand: Section */
#define ET_PARSER_SECTION			":DP-Attr unbekannt"

#define EC_PARSER_DATA				20	/* Fehler im Parser-Zustand: Data */
#define ET_PARSER_DATA				":DP-Attr unbekannt"

#define EC_NO_PGLOBALS				21	/* Fehler, da kein gültiger pGlobals-Pointer */
#define ET_NO_PGLOBALS				":kein pGlobals"

#define EC_PORT_ALREADY_EXISTS		22	/* Fehler, da Port bereits vergeben */
#define ET_PORT_ALREADY_EXISTS		":Port bereits vorh."

#define EC_TIMEOUT_ALREADY_EXISTS	23	/* Fehler, da Tiemout bereits vergeben */
#define ET_TIMEOUT_ALREADY_EXISTS	":Timeout bereits vorh"

#define EC_TYPE_ALREADY_EXIST		24	/* Fehler, da Datentyp bereits existiert */
#define ET_TYPE_ALREADY_EXIST		":TYP Name falsch"

#define EC_TYPE_NO_INVALID			25	/* Fehler, da Datenpunkt bereits existiert */
#define ET_TYPE_NO_INVALID			":TYP Nr falsch"

#define EC_POINT_ALREADY_EXIST		26	/* Fehler, da Datenpunkt bereits existiert */
#define ET_POINT_ALREADY_EXIST		":Dp bereits vorhanden"

#define EC_NO_LINK_FUB_DBSERV		27	/* Fehler, da Datenpunkt bereits existiert */
#define ET_NO_LINK_FUB_DBSERV		"Verkettung unvollständig"

#define EC_NO_LINK_DBSERV_FUB		28	/* Fehler, da Datenpunkt bereits existiert */
#define ET_NO_LINK_DBSERV_FUB		"Verkettung unvollständig"

#define EC_NO_TIMESTAMP_FUB			29	/* Fehler, da Datenpunkt bereits existiert */
#define ET_NO_TIMESTAMP_FUB			"Fub ohne Zeitstempel"

#define EC_BUF_EVENTS				30	/* Fehler, da Datenpunkt bereits existiert */
#define ET_BUF_EVENTS				"Archiv EventAnz="

#define EC_MEM_EVENTS				31	/* Fehler, da Datenpunkt bereits existiert */
#define ET_MEM_EVENTS				"Archiv Mem="

#define EC_BOOL_PREFIX				50
#define ET_BOOL_PREFIX				"BOOL"

#define EC_BOOL_TS_PREFIX			51
#define ET_BOOL_TS_PREFIX			"BOOL_TS"

#define EC_USINT_PREFIX				52
#define ET_USINT_PREFIX				"USINT"

#define EC_USINT_TS_PREFIX			53
#define ET_USINT_TS_PREFIX			"USINT_TS"

#define EC_UINT_PREFIX				54
#define ET_UINT_PREFIX				"UINT"

#define EC_INT_PREFIX				55
#define ET_INT_PREFIX				"INT"

#define EC_UDINT_PREFIX				56
#define ET_UDINT_PREFIX				"UDINT"

#define EC_DINT_PREFIX				57
#define ET_DINT_PREFIX				"DINT"

#define EC_MAX						60	/* Anzahl Fehlereinträge */

/***********************************************************************/
/* Datentypdeklaration                                                 */
/***********************************************************************/

typedef plcbit BIT;			/* Datentyp BIT */

/* -------------------------------- */
/* Datentypen für Item-Deskriptoren */
/* -------------------------------- */
typedef struct {
	unsigned short	offItem;
	unsigned short	lenItem;
	unsigned char	sItem;
	unsigned char	tsItem;
	unsigned char	FileBuffer;
	unsigned char	idTypeItem;
	unsigned char	*pNameItem;
} ITEM_DESC;

/* ------------------------------- */
/* Datentypen für Typ-Deskriptoren */
/* ------------------------------- */
typedef struct {
	unsigned short	dbsType;
	unsigned short	sizeType;
	unsigned short	sizeIntType;
	unsigned char	*pTypeName;
	unsigned short	countItem;
	unsigned short	countTimeItem;
	ITEM_DESC		*pItemDesc;
	unsigned short	countRelatedPoints;
	unsigned char	FileBuffer;
	unsigned char	ModeFileBuffer;
	unsigned long	EventFileBuffer;
	unsigned long	SizeFileBuffer;
} TYPE_DESC;

/* --------------------------------- */
/* Datentypen für Punkt-Deskriptoren */
/* --------------------------------- */
typedef struct {
	unsigned short	dbsUnit;
	unsigned short	dbsType;
	unsigned short	dbsPoint;
	unsigned char	*pPointName;
} POINT_DESC;

/* -------------------------------------- */
/* Datentypen für Fubinstanz-Deskriptoren */
/* -------------------------------------- */
typedef struct {
	unsigned short	dbsUnit;
	unsigned short	dbsType;
	unsigned short	dbsPoint;
	unsigned short	dbsItem;
	unsigned char	*pFubInstance;
} FUB_DESC;

/* ------------------------- */
/* Datentypen für Eventpipes */
/* ------------------------- */
typedef struct {
	UDINT	countEvent;
	UDINT	firstEvent;
	UDINT	lastEvent;
} PIPE_EVENT_STATE;

typedef struct {
	PIPE_EVENT_STATE	stateEvent;
	UINT	pipe_entry;
	UINT	pipe_size;
	UINT	pipe_level;
	USINT*	pPipeData;
	UINT	iPipeRead;
	UINT	iPipeWrite;
} EVENT_PIPE_HEADER;

typedef struct {
	USINT	linkstate;
	USINT	eventtype;
	UINT	unit;
	UINT	device;
	UINT	type;
	UINT	point;
	UINT	item;
	UDINT	length;
	USINT*	pData;
} EVENT_PIPE_DATA;

typedef struct {
	EVENT_PIPE_HEADER*	pEventPipeHeaderWrite[2];
	EVENT_PIPE_HEADER*	pEventPipeHeaderRead;
	UINT				BufferEventIndex;
	UINT				BufferFileIndex;
	BOOL				WriteDataBusy;
	BOOL				ReadDataBusy;
	BOOL				GetEventsFromReadPipe;

	UDINT				xlength_pipe_next;
/*
	BOOL				WriteToFile;
	USINT				ModeFileBuffer;
	UDINT				SizeFileBuffer;
*/
	USINT				FileDevice[32];
	USINT				FileName[32];
	UDINT				fileIdent;
	UDINT				fileLen;
	UDINT				fileOffsetWrite;
	UDINT				fileOffsetRead;
	UINT				fileStep;
	UINT				fileState;
	UINT				fileSysError;

	FileOpen_typ		iFileOpen;
	FileCreate_typ		iFileCreate;
	FileWrite_typ		iFileWrite;
	FileRead_typ		iFileRead;
	FileClose_typ		iFileClose;
	FileDelete_typ		iFileDelete;
} EVENT_PIPE_INSTANCE;

typedef struct {
	BOOL					WriteToFile;
	USINT					ModeFileBuffer;
	UDINT					SizeFileBuffer;
	EVENT_PIPE_INSTANCE*	pEventPipeInstance;
} ACCESS_EVENT_PIPE;

typedef struct {
	UINT	pipe_entry;
	UINT	pipe_size;
	UINT	pipe_level;
	USINT*	pPipeData;
	UINT	iPipeRead;
	UINT	iPipeWrite;

	UDINT	TickCount;
	UINT	iLastPipeRead;
	UINT	unit;
	UINT	device;
	UINT	type;
	UINT	point;
	UINT	item;
} WRITE_PIPE_HEADER;

typedef struct {
	USINT	linkstate;
	USINT	eventtype;
	UINT	unit;
	UINT	device;
	UINT	type;
	UINT	point;
	UINT	item;
	UDINT	length;
	USINT*	pData;
} WRITE_PIPE_DATA;

typedef struct {
	WRITE_PIPE_HEADER*	pWritePipeHeader;
	UDINT				length_pipe_next;
} ACCESS_WRITE_PIPE;

/* ---------------------------------------- */
/* Datentypen für Zugriff auf Prozessabbild */
/* ---------------------------------------- */
typedef struct {
	unsigned char	ItemEventState;
} ITEM_EVENT_STATE;

typedef struct {
	UDINT	noEvent;
} POINT_EVENT_STATE;

typedef struct {
	UDINT	countEvent;
} TYPE_EVENT_STATE;

typedef struct {
	UDINT	countEvent;
} UNIT_EVENT_STATE;

typedef struct {
	UDINT	countEvent;
} SERVER_EVENT_STATE;

/* ---------------------------------------- */
/* Datentypen für Zugriff auf Prozessabbild */
/* ---------------------------------------- */
typedef USINT	ACCESS_ITEM_VALID;
typedef USINT	ACCESS_ITEM_EVENT_LINK;
typedef USINT	ACCESS_ITEM_WRITE_LINK;
typedef UDINT	ACCESS_ITEM_WRITE_HANDLE;
typedef USINT	ACCESS_ITEM_RELEASE;

typedef USINT	ACCESS_ITEM_EVENT_STATE;

typedef USINT*	ACCESS_FUB_INSTANCE;

typedef unsigned char	ACCESS_DATA;

typedef struct {
	unsigned short	countItem;
	ACCESS_DATA		*pAccessData;
} ACCESS_POINT;

typedef struct {
	unsigned short	countPoint;
	ACCESS_POINT	*pAccessPoint;

	unsigned long	offExtern;
	unsigned long	lenExtern;

	unsigned long	offIntern;
	unsigned long	lenIntern;

	unsigned long	offiExtern;
	unsigned long	leniExtern;
	unsigned long	leniExternAlign;
	unsigned long	leniExternNext;		/* Abstand für Instanzen */

	unsigned long	offValid;
	unsigned long	lenValid;
	unsigned long	lenValidAlign;		/* Abstand für Items */

	unsigned long	offTime;
	unsigned long	lenTime;
	unsigned long	lenTimeAlign;		/* Abstand für Items */

	unsigned long	offiTime;
	unsigned long	leniTime;
	unsigned long	leniTimeAlign;		/* Abstand für Items */
	unsigned long	leniTimeNext;		/* Abstand für Instanzen */

	unsigned long	offWritelink;
	unsigned long	lenWritelink;
	unsigned long	lenWritelinkAlign;	/* Abstand für Items */

	unsigned long	offWritehandle;
	unsigned long	lenWritehandle;
	unsigned long	lenWritehandleAlign;/* Abstand für Items */

	unsigned long	offiEventlink;
	unsigned long	leniEventlink;
	unsigned long	leniEventlinkAlign;	/* Abstand für Items */
	unsigned long	leniEventlinkNext;	/* Abstand für Instanzen */

	unsigned long	offiReleasestream;
	unsigned long	leniReleasestream;
	unsigned long	leniReleasestreamAlign;	/* Abstand für Items */
	unsigned long	leniReleasestreamNext;	/* Abstand für Instanzen */

	unsigned long	offiHyst;
	unsigned long	leniHyst;
	unsigned long	leniHystAlign;
	unsigned long	leniHystNext;		/* Abstand für Instanzen */

	unsigned long	offiEvent;
	unsigned long	leniEvent;
	unsigned long	leniEventAlign;		/* Abstand für Items */
	unsigned long	leniEventNext;		/* Abstand für Instanzen */

	unsigned long	offFubInstance;
	unsigned long	lenFubInstance;
	unsigned long	lenFubInstanceAlign;
} ACCESS_TYPE;

typedef struct {
	unsigned short	countType;
	ACCESS_TYPE*	pAccessType;
} ACCESS_UNIT;

typedef struct {
	unsigned short		countEventInstance;
	unsigned short		countWriteInstance;
	unsigned short		countType;
	unsigned short		countUnit;
	ACCESS_UNIT*		pAccessUnit;
	TYPE_DESC*			pAccessTypeDesc;
	POINT_DESC*			pAccessPointDesc;
	unsigned short		noDevice;
	UNIT_EVENT_STATE*	pUnitEventState;
	ACCESS_EVENT_PIPE*	pAccessEventPipe;
	ACCESS_WRITE_PIPE*	pAccessWritePipe;
	unsigned short		PortNumber;
	unsigned short		TimeoutValue;
	unsigned long		TimeOutWritePipe;
	unsigned long		TickCount;
} ACCESS_SERVER;

/***********************************************************************/
/* DbServ-Funktionen                                                  */
/***********************************************************************/
unsigned char IsANumber(unsigned char *pData);
int ltoa(long value, char *buffer);
int ultoa(unsigned long value, char *buffer);

/*============================= Ende der Datei ==============================*/

/* ------------------- */
/* Fehler-Definitionen */
/* ------------------- */
#define cEC_OK								0

#define cEC_INVALID_SERVER					1000
#define cEC_NOT_READY_SERVER				1010
#define cEC_INVALID_INSTANCE				1001
#define cEC_INVALID_UNIT					1002
#define cEC_INVALID_DEVICE					1003
#define cEC_INVALID_TYPE					1004
#define cEC_INVALID_POINT					1005
#define cEC_INVALID_ITEM					1006
#define cEC_INVALID_VALUE					1007

#define cEC_INVALID_TYPE_FOR_HYST			1100
#define cEC_INVALID_POINT_FOR_HYST			1101

#define cEC_NO_DATA_IN_EVENTBUFFER			1200
#define cEC_EVENTBUFFER_TO_SMALL			1201

#define cEC_ITEM_ALREADY_LINKED				1300
#define cEC_ITEM_ALREADY_UNLINKED			1301
#define cEC_ITEM_NO_TIMESTAMP				1302
#define cEC_ITEM_ALREADY_LINKED_FILE_BUFFER	1303
#define cEC_ITEM_NOT_UNLINKED_FILE_BUFFER	1304

#define cEC_INVALID_LENGTH					1400
#define cEC_INVALID_HANDLE					1401

#define cEC_ITEM_NOT_WRITEABLE				1500
#define cEC_NO_DATA_IN_WRITEBUFFER			1501
#define cEC_WRITE_PIPE_FULL					1502

#define cEC_FUB_NOT_LINKED_DBSERV			1600
#define cEC_DBSERV_NOT_LINKED_FUB			1601

#define cEC_FUB_WITHOUT_TIMESTAMP			1700

/* ------------------- */
/* Status-Definitionen */
/* ------------------- */
enum {	cITEM_UNLINKED,
		cITEM_LINKED_WITHOUT_TIMESTAMP,
		cITEM_LINKED_WITH_TIMESTAMP	};

/* ----------------------- */
/* Funktionen für Brserver */
/* ----------------------- */
UINT GetIdBrServer (void **pidBrServer, UINT *pbrstate);
UINT GetPortNumber (void *idBrServer, UINT *pPortNumber);
UINT GetTimeoutValue (void *idBrServer, UINT *pTimeoutValue);
UINT GetEventInstanceInfo (void *idBrServer, UINT *pEventInstance);
UINT GetWriteInstanceInfo (void *idBrServer, UINT *pWriteInstance);
UINT GetTypeInfo (void *idBrServer, UINT *ptype);
UINT GetItemInfo (void *idBrServer, UINT instance,
					UINT unit, UINT device, UINT type, UINT point, UINT item,
					USINT** ppData_extern,		UDINT* plength_extern,
					USINT** ppData_intern,		UDINT* plength_intern,
					USINT** ppData_iextern,		UDINT* plength_iextern,
					USINT** ppData_valid,		UDINT* plength_valid,
					USINT** ppData_time,		UDINT* plength_time,
					USINT** ppData_itime,		UDINT* plength_itime,
					USINT** ppData_writelink,	UDINT* plength_writelink,
					USINT** ppData_ieventlink,	UDINT* plength_ieventlink,
					USINT** ppData_ihyst,		UDINT* plength_ihyst,
					USINT** ppData_ievent,		UDINT* plength_ievent);
UINT GetEventLinkInfo (void *idBrServer,
						UINT unit, UINT device, UINT type, UINT point, UINT item,
						UINT *pcountInstanceAll, UINT *pcountInstanceNoTimestamp, UINT *pcountInstanceTimestamp, USINT *ptsItem);
UINT GetEventPipeInfo (void *idBrServer, UINT instance, UINT type,
						UINT *pipe_entry, UINT *pipe_level_abs, USINT *pipe_level_rel);
UINT GetWritePipeInfo (void *idBrServer, UINT instance,
						UINT *pipe_entry, UINT *pipe_level_abs, USINT *pipe_level_rel);
UINT GetFubInstance (void *idBrServer,
						UINT unit, UINT device, UINT type, UINT point, UINT item,
						USINT **ppFubInstance);
UINT LinkEventInstance (void *idBrServer, UINT instance);
UINT UnlinkEventInstance (void *idBrServer, UINT instance);
UINT UnlinkEventInstanceWithoutFileBuffer (void *idBrServer, UINT instance);
UINT LinkEventUnit (void *idBrServer, UINT instance,
					UINT unit);
UINT UnLinkEventUnit (void *idBrServer, UINT instance,
						UINT unit);
UINT LinkEventDevice (void *idBrServer, UINT instance,
						UINT unit, UINT device);
UINT UnLinkEventDevice (void *idBrServer, UINT instance,
						UINT unit, UINT device);
UINT LinkEventType (void *idBrServer, UINT instance,
					UINT unit, UINT device, UINT type);
UINT UnlinkEventType (void *idBrServer, UINT instance,
						UINT unit, UINT device, UINT type);
UINT LinkEventItem (void *idBrServer, UINT instance,
					UINT unit, UINT device, UINT type, UINT point, UINT item,
					USINT timestamp);
UINT UnlinkEventItem (void *idBrServer, UINT instance,
						UINT unit, UINT device, UINT type, UINT point, UINT item);
UINT UnlinkEventItemWithoutFileBuffer (void *idBrServer, UINT instance,
										UINT unit, UINT device, UINT type, UINT point, UINT item);
UINT SetHystItem (void *idBrServer, UINT instance,
					UINT unit, UINT device, UINT type, UINT point, UINT item,
					USINT* pValue, UDINT lengthValue);
UINT SetValueItem (void *idBrServer,
					UINT unit, UINT device, UINT type, UINT point, UINT item,
					USINT* pValue, UDINT lengthValue,
					RTCtime_typ RTCTime, USINT setTimeStampNow,
					USINT enableEvent);
UINT GetValueItem (void *idBrServer, UINT instance,
					UINT unit, UINT device, UINT type, UINT point, UINT item,
					USINT** ppData_extern, UDINT* plength_extern,
					USINT** ppData_time, UDINT* plength_time);
UINT GetValueItemNoUpdate (void *idBrServer,
							UINT unit, UINT device, UINT type, UINT point, UINT item,
							USINT** ppData_extern, UDINT* plength_extern,
							USINT** ppData_time, UDINT* plength_time);
UINT SetEventItem (void *idBrServer, UINT instance,
					UINT unit, UINT device, UINT type, UINT point, UINT item,
					USINT *pValue, UINT lengthValue,
					USINT eventtype, USINT *pDataExtern, RTCtime_typ RTCTime);
UINT SetEventItemStream (void *idBrServer,
							UINT unit, UINT device, UINT type, UINT point, UINT item,
							USINT *pValue, UDINT lengthValue,
							USINT *pFlag,
							RTCtime_typ RTCTime, USINT setTimeStampNow,
							USINT enableEvent);
UINT ReleaseEventItemStream (void *idBrServer, UINT instance,
								UINT unit, UINT device, UINT type, UINT point, UINT item);
UINT GetEventItem (void *idBrServer, UINT instance,
					UINT type, USINT *pEventBuffer, UDINT lengthEventBuffer,
					UDINT* pLength, UDINT *pLengthTimeStamp);
UINT WorkEvent (void *idBrServer);
UINT LinkWriteInstance (void *idBrServer, UINT instance);
UINT UnlinkWriteInstance (void *idBrServer, UINT instance);
UINT LinkWriteUnit (void *idBrServer, UINT instance,
					UINT unit);
UINT UnlinkWriteUnit (void *idBrServer, UINT instance,
						UINT unit);
UINT LinkWriteDevice (void *idBrServer, UINT instance,
						UINT unit, UINT device);
UINT UnlinkWriteDevice (void *idBrServer, UINT instance,
						UINT unit, UINT device);
UINT LinkWriteType (void *idBrServer, UINT instance,
					UINT unit, UINT device, UINT type);
UINT UnlinkWriteType (void *idBrServer, UINT instance,
						UINT unit, UINT device, UINT type);
UINT LinkWriteItem (void *idBrServer, UINT instance,
					UINT unit, UINT device, UINT type, UINT point, UINT item,
					UDINT handle);
UINT UnlinkWriteItem (void *idBrServer, UINT instance,
						UINT unit, UINT device, UINT type, UINT point, UINT item);
UINT SetWriteItem (void *dBrServer,
					UINT unit, UINT device, UINT type, UINT point, UINT item,
					USINT* pValue, UDINT lengthValue);
UINT ScanWriteItem (void *idBrServer, UINT instance,
					USINT* pWriteBuffer, UDINT lengthWriteBuffer,
					UDINT* pLength, UDINT* pLengthTimeStamp);
UINT GetWriteItem (void *idBrServer, UINT instance,
					USINT* pWriteBuffer, UDINT lengthWriteBuffer,
					UDINT* pLength, UDINT* pLengthTimeStamp);
UINT CopyPipeToFile (void *idBrServer);

/*============================= Ende der Datei ==============================*/
```
